    CONST robtarget T677:=[[56.500013,76.537078,6.249631],[1.000000,0.000000,0.000000,0.000000],[0,0,-1,0],[9E+09,9E+09,9E+09,9E+09,9E+09,9E+09]];
    CONST robtarget T678:=[[58.000019,76.384788,6.249631],[1.000000,0.000000,0.000000,0.000000],[0,0,-1,0],[9E+09,9E+09,9E+09,9E+09,9E+09,9E+09]];
    CONST robtarget T679:=[[58.000019,35.406248,6.249631],[1.000000,0.000000,0.000000,0.000000],[0,0,-1,0],[9E+09,9E+09,9E+09,9E+09,9E+09,9E+09]];
    CONST robtarget T680:=[[59.500025,35.473840,6.249631],[1.000000,0.000000,0.000000,0.000000],[0,0,-1,0],[9E+09,9E+09,9E+09,9E+09,9E+09,9E+09]];
    CONST robtarget T681:=[[59.500025,76.264330,6.249631],[1.000000,0.000000,0.000000,0.000000],[0,0,-1,0],[9E+09,9E+09,9E+09,9E+09,9E+09,9E+09]];
    CONST robtarget T682:=[[61.000031,76.089981,6.249631],[1.000000,0.000000,0.000000,0.000000],[0,0,-1,0],[9E+09,9E+09,9E+09,9E+09,9E+09,9E+09]];
    CONST robtarget T683:=[[61.000031,35.612525,6.249631],[1.000000,0.000000,0.000000,0.000000],[0,0,-1,0],[9E+09,9E+09,9E+09,9E+09,9E+09,9E+09]];
    CONST robtarget T684:=[[62.500037,35.829098,6.249631],[1.000000,0.000000,0.000000,0.000000],[0,0,-1,0],[9E+09,9E+09,9E+09,9E+09,9E+09,9E+09]];
    CONST robtarget T685:=[[62.500037,75.849994,6.249631],[1.000000,0.000000,0.000000,0.000000],[0,0,-1,0],[9E+09,9E+09,9E+09,9E+09,9E+09,9E+09]];
    CONST robtarget T686:=[[64.000043,75.305600,6.249631],[1.000000,0.000000,0.000000,0.000000],[0,0,-1,0],[9E+09,9E+09,9E+09,9E+09,9E+09,9E+09]];
    CONST robtarget T687:=[[64.000043,36.214677,6.249631],[1.000000,0.000000,0.000000,0.000000],[0,0,-1,0],[9E+09,9E+09,9E+09,9E+09,9E+09,9E+09]];
    CONST robtarget T688:=[[65.500049,36.567546,6.249631],[1.000000,0.000000,0.000000,0.000000],[0,0,-1,0],[9E+09,9E+09,9E+09,9E+09,9E+09,9E+09]];
    CONST robtarget T689:=[[65.500049,74.486668,6.249631],[1.000000,0.000000,0.000000,0.000000],[0,0,-1,0],[9E+09,9E+09,9E+09,9E+09,9E+09,9E+09]];
    CONST robtarget T690:=[[67.000055,73.456702,6.249631],[1.000000,0.000000,0.000000,0.000000],[0,0,-1,0],[9E+09,9E+09,9E+09,9E+09,9E+09,9E+09]];
    CONST robtarget T691:=[[67.000055,37.225942,6.249631],[1.000000,0.000000,0.000000,0.000000],[0,0,-1,0],[9E+09,9E+09,9E+09,9E+09,9E+09,9E+09]];
    CONST robtarget T692:=[[68.500061,37.908304,6.249631],[1.000000,0.000000,0.000000,0.000000],[0,0,-1,0],[9E+09,9E+09,9E+09,9E+09,9E+09,9E+09]];
    CONST robtarget T693:=[[68.500061,72.303444,6.249631],[1.000000,0.000000,0.000000,0.000000],[0,0,-1,0],[9E+09,9E+09,9E+09,9E+09,9E+09,9E+09]];
    CONST robtarget T694:=[[70.000067,70.867702,6.249631],[1.000000,0.000000,0.000000,0.000000],[0,0,-1,0],[9E+09,9E+09,9E+09,9E+09,9E+09,9E+09]];
    CONST robtarget T695:=[[70.000067,38.836205,6.249631],[1.000000,0.000000,0.000000,0.000000],[0,0,-1,0],[9E+09,9E+09,9E+09,9E+09,9E+09,9E+09]];
    CONST robtarget T696:=[[71.500073,39.891103,6.249631],[1.000000,0.000000,0.000000,0.000000],[0,0,-1,0],[9E+09,9E+09,9E+09,9E+09,9E+09,9E+09]];
    CONST robtarget T697:=[[71.500073,69.078100,6.249631],[1.000000,0.000000,0.000000,0.000000],[0,0,-1,0],[9E+09,9E+09,9E+09,9E+09,9E+09,9E+09]];
    CONST robtarget T698:=[[73.000079,66.945059,6.249631],[1.000000,0.000000,0.000000,0.000000],[0,0,-1,0],[9E+09,9E+09,9E+09,9E+09,9E+09,9E+09]];
    CONST robtarget T699:=[[73.000079,41.103881,6.249631],[1.000000,0.000000,0.000000,0.000000],[0,0,-1,0],[9E+09,9E+09,9E+09,9E+09,9E+09,9E+09]];
    CONST robtarget T700:=[[74.500085,42.494022,6.249631],[1.000000,0.000000,0.000000,0.000000],[0,0,-1,0],[9E+09,9E+09,9E+09,9E+09,9E+09,9E+09]];
    CONST robtarget T701:=[[74.500085,64.388687,6.249631],[1.000000,0.000000,0.000000,0.000000],[0,0,-1,0],[9E+09,9E+09,9E+09,9E+09,9E+09,9E+09]];
    CONST robtarget T702:=[[76.000091,60.363543,6.249631],[1.000000,0.000000,0.000000,0.000000],[0,0,-1,0],[9E+09,9E+09,9E+09,9E+09,9E+09,9E+09]];
    CONST robtarget T703:=[[76.000091,44.225148,6.249631],[1.000000,0.000000,0.000000,0.000000],[0,0,-1,0],[9E+09,9E+09,9E+09,9E+09,9E+09,9E+09]];
    CONST robtarget T704:=[[77.500097,47.712288,6.249631],[1.000000,0.000000,0.000000,0.000000],[0,0,-1,0],[9E+09,9E+09,9E+09,9E+09,9E+09,9E+09]];
    CONST robtarget T705:=[[77.500097,54.837844,6.249631],[1.000000,0.000000,0.000000,0.000000],[0,0,-1,0],[9E+09,9E+09,9E+09,9E+09,9E+09,9E+09]];
    CONST robtarget T706:=[[77.500097,46.672683,6.749641],[1.000000,0.000000,0.000000,0.000000],[0,0,-1,0],[9E+09,9E+09,9E+09,9E+09,9E+09,9E+09]];
    CONST robtarget T707:=[[77.500097,56.264594,6.749641],[1.000000,0.000000,0.000000,0.000000],[0,0,-1,0],[9E+09,9E+09,9E+09,9E+09,9E+09,9E+09]];
    CONST robtarget T708:=[[77.500097,46.672683,6.749641],[1.000000,0.000000,0.000000,0.000000],[0,0,-1,0],[9E+09,9E+09,9E+09,9E+09,9E+09,9E+09]];
    CONST robtarget T709:=[[77.500097,56.264594,6.749641],[1.000000,0.000000,0.000000,0.000000],[0,0,-1,0],[9E+09,9E+09,9E+09,9E+09,9E+09,9E+09]];
    CONST robtarget T710:=[[76.000091,60.945739,6.749641],[1.000000,0.000000,0.000000,0.000000],[0,0,-1,0],[9E+09,9E+09,9E+09,9E+09,9E+09,9E+09]];
    CONST robtarget T711:=[[76.000091,43.718418,6.749641],[1.000000,0.000000,0.000000,0.000000],[0,0,-1,0],[9E+09,9E+09,9E+09,9E+09,9E+09,9E+09]];
    CONST robtarget T712:=[[74.500085,42.018319,6.749641],[1.000000,0.000000,0.000000,0.000000],[0,0,-1,0],[9E+09,9E+09,9E+09,9E+09,9E+09,9E+09]];
    CONST robtarget T713:=[[74.500085,64.686211,6.749641],[1.000000,0.000000,0.000000,0.000000],[0,0,-1,0],[9E+09,9E+09,9E+09,9E+09,9E+09,9E+09]];
    CONST robtarget T714:=[[73.000079,67.110705,6.749641],[1.000000,0.000000,0.000000,0.000000],[0,0,-1,0],[9E+09,9E+09,9E+09,9E+09,9E+09,9E+09]];
    CONST robtarget T715:=[[73.000079,40.678790,6.749641],[1.000000,0.000000,0.000000,0.000000],[0,0,-1,0],[9E+09,9E+09,9E+09,9E+09,9E+09,9E+09]];
    CONST robtarget T716:=[[71.500073,39.412409,6.749641],[1.000000,0.000000,0.000000,0.000000],[0,0,-1,0],[9E+09,9E+09,9E+09,9E+09,9E+09,9E+09]];
    CONST robtarget T717:=[[71.500073,69.236494,6.749641],[1.000000,0.000000,0.000000,0.000000],[0,0,-1,0],[9E+09,9E+09,9E+09,9E+09,9E+09,9E+09]];
    CONST robtarget T718:=[[70.000067,71.090670,6.749641],[1.000000,0.000000,0.000000,0.000000],[0,0,-1,0],[9E+09,9E+09,9E+09,9E+09,9E+09,9E+09]];
    CONST robtarget T719:=[[70.000067,38.385338,6.749641],[1.000000,0.000000,0.000000,0.000000],[0,0,-1,0],[9E+09,9E+09,9E+09,9E+09,9E+09,9E+09]];
    CONST robtarget T720:=[[68.500061,37.449765,6.749641],[1.000000,0.000000,0.000000,0.000000],[0,0,-1,0],[9E+09,9E+09,9E+09,9E+09,9E+09,9E+09]];
    CONST robtarget T721:=[[68.500061,72.617147,6.749641],[1.000000,0.000000,0.000000,0.000000],[0,0,-1,0],[9E+09,9E+09,9E+09,9E+09,9E+09,9E+09]];
    CONST robtarget T722:=[[67.000055,73.796696,6.749641],[1.000000,0.000000,0.000000,0.000000],[0,0,-1,0],[9E+09,9E+09,9E+09,9E+09,9E+09,9E+09]];
    CONST robtarget T723:=[[67.000055,36.779468,6.749641],[1.000000,0.000000,0.000000,0.000000],[0,0,-1,0],[9E+09,9E+09,9E+09,9E+09,9E+09,9E+09]];
    CONST robtarget T724:=[[65.500049,36.130056,6.749641],[1.000000,0.000000,0.000000,0.000000],[0,0,-1,0],[9E+09,9E+09,9E+09,9E+09,9E+09,9E+09]];
    CONST robtarget T725:=[[65.500049,74.800360,6.749641],[1.000000,0.000000,0.000000,0.000000],[0,0,-1,0],[9E+09,9E+09,9E+09,9E+09,9E+09,9E+09]];
    CONST robtarget T726:=[[64.000043,75.578750,6.749641],[1.000000,0.000000,0.000000,0.000000],[0,0,-1,0],[9E+09,9E+09,9E+09,9E+09,9E+09,9E+09]];
    CONST robtarget T727:=[[64.000043,35.777188,6.749641],[1.000000,0.000000,0.000000,0.000000],[0,0,-1,0],[9E+09,9E+09,9E+09,9E+09,9E+09,9E+09]];
    CONST robtarget T728:=[[62.500037,35.412563,6.749641],[1.000000,0.000000,0.000000,0.000000],[0,0,-1,0],[9E+09,9E+09,9E+09,9E+09,9E+09,9E+09]];
    CONST robtarget T729:=[[62.500037,76.134604,6.749641],[1.000000,0.000000,0.000000,0.000000],[0,0,-1,0],[9E+09,9E+09,9E+09,9E+09,9E+09,9E+09]];
    CONST robtarget T730:=[[61.000031,76.390171,6.749641],[1.000000,0.000000,0.000000,0.000000],[0,0,-1,0],[9E+09,9E+09,9E+09,9E+09,9E+09,9E+09]];
    CONST robtarget T731:=[[61.000031,35.224978,6.749641],[1.000000,0.000000,0.000000,0.000000],[0,0,-1,0],[9E+09,9E+09,9E+09,9E+09,9E+09,9E+09]];
    CONST robtarget T732:=[[59.500025,35.088916,6.749641],[1.000000,0.000000,0.000000,0.000000],[0,0,-1,0],[9E+09,9E+09,9E+09,9E+09,9E+09,9E+09]];
    CONST robtarget T733:=[[59.500025,76.568137,6.749641],[1.000000,0.000000,0.000000,0.000000],[0,0,-1,0],[9E+09,9E+09,9E+09,9E+09,9E+09,9E+09]];
    CONST robtarget T734:=[[58.000019,76.697078,6.749641],[1.000000,0.000000,0.000000,0.000000],[0,0,-1,0],[9E+09,9E+09,9E+09,9E+09,9E+09,9E+09]];
    CONST robtarget T735:=[[58.000019,35.030106,6.749641],[1.000000,0.000000,0.000000,0.000000],[0,0,-1,0],[9E+09,9E+09,9E+09,9E+09,9E+09,9E+09]];
    CONST robtarget T736:=[[56.500013,34.993140,6.749641],[1.000000,0.000000,0.000000,0.000000],[0,0,-1,0],[9E+09,9E+09,9E+09,9E+09,9E+09,9E+09]];
    CONST robtarget T737:=[[56.500013,76.858293,6.749641],[1.000000,0.000000,0.000000,0.000000],[0,0,-1,0],[9E+09,9E+09,9E+09,9E+09,9E+09,9E+09]];
    CONST robtarget T738:=[[55.000007,76.963959,6.749641],[1.000000,0.000000,0.000000,0.000000],[0,0,-1,0],[9E+09,9E+09,9E+09,9E+09,9E+09,9E+09]];
    CONST robtarget T739:=[[55.000007,34.997342,6.749641],[1.000000,0.000000,0.000000,0.000000],[0,0,-1,0],[9E+09,9E+09,9E+09,9E+09,9E+09,9E+09]];
    CONST robtarget T740:=[[53.500001,34.993140,6.749641],[1.000000,0.000000,0.000000,0.000000],[0,0,-1,0],[9E+09,9E+09,9E+09,9E+09,9E+09,9E+09]];
    CONST robtarget T741:=[[53.500001,76.858293,6.749641],[1.000000,0.000000,0.000000,0.000000],[0,0,-1,0],[9E+09,9E+09,9E+09,9E+09,9E+09,9E+09]];
    CONST robtarget T742:=[[51.999995,76.697078,6.749641],[1.000000,0.000000,0.000000,0.000000],[0,0,-1,0],[9E+09,9E+09,9E+09,9E+09,9E+09,9E+09]];
    CONST robtarget T743:=[[51.999995,35.030107,6.749641],[1.000000,0.000000,0.000000,0.000000],[0,0,-1,0],[9E+09,9E+09,9E+09,9E+09,9E+09,9E+09]];
    CONST robtarget T744:=[[50.499989,35.088916,6.749641],[1.000000,0.000000,0.000000,0.000000],[0,0,-1,0],[9E+09,9E+09,9E+09,9E+09,9E+09,9E+09]];
    CONST robtarget T745:=[[50.499989,76.568136,6.749641],[1.000000,0.000000,0.000000,0.000000],[0,0,-1,0],[9E+09,9E+09,9E+09,9E+09,9E+09,9E+09]];
    CONST robtarget T746:=[[48.999983,76.390167,6.749641],[1.000000,0.000000,0.000000,0.000000],[0,0,-1,0],[9E+09,9E+09,9E+09,9E+09,9E+09,9E+09]];
    CONST robtarget T747:=[[48.999983,35.224979,6.749641],[1.000000,0.000000,0.000000,0.000000],[0,0,-1,0],[9E+09,9E+09,9E+09,9E+09,9E+09,9E+09]];
    CONST robtarget T748:=[[47.499977,35.412564,6.749641],[1.000000,0.000000,0.000000,0.000000],[0,0,-1,0],[9E+09,9E+09,9E+09,9E+09,9E+09,9E+09]];
    CONST robtarget T749:=[[47.499977,76.134597,6.749641],[1.000000,0.000000,0.000000,0.000000],[0,0,-1,0],[9E+09,9E+09,9E+09,9E+09,9E+09,9E+09]];
    CONST robtarget T750:=[[45.999971,75.578745,6.749641],[1.000000,0.000000,0.000000,0.000000],[0,0,-1,0],[9E+09,9E+09,9E+09,9E+09,9E+09,9E+09]];
    CONST robtarget T751:=[[45.999971,35.777189,6.749641],[1.000000,0.000000,0.000000,0.000000],[0,0,-1,0],[9E+09,9E+09,9E+09,9E+09,9E+09,9E+09]];
    CONST robtarget T752:=[[44.499965,36.130058,6.749641],[1.000000,0.000000,0.000000,0.000000],[0,0,-1,0],[9E+09,9E+09,9E+09,9E+09,9E+09,9E+09]];
    CONST robtarget T753:=[[44.499965,74.800359,6.749641],[1.000000,0.000000,0.000000,0.000000],[0,0,-1,0],[9E+09,9E+09,9E+09,9E+09,9E+09,9E+09]];
    CONST robtarget T754:=[[42.999959,73.796696,6.749641],[1.000000,0.000000,0.000000,0.000000],[0,0,-1,0],[9E+09,9E+09,9E+09,9E+09,9E+09,9E+09]];
    CONST robtarget T755:=[[42.999959,36.779470,6.749641],[1.000000,0.000000,0.000000,0.000000],[0,0,-1,0],[9E+09,9E+09,9E+09,9E+09,9E+09,9E+09]];
    CONST robtarget T756:=[[41.499953,37.449766,6.749641],[1.000000,0.000000,0.000000,0.000000],[0,0,-1,0],[9E+09,9E+09,9E+09,9E+09,9E+09,9E+09]];
    CONST robtarget T757:=[[41.499953,72.617146,6.749641],[1.000000,0.000000,0.000000,0.000000],[0,0,-1,0],[9E+09,9E+09,9E+09,9E+09,9E+09,9E+09]];
    CONST robtarget T758:=[[39.999947,71.090670,6.749641],[1.000000,0.000000,0.000000,0.000000],[0,0,-1,0],[9E+09,9E+09,9E+09,9E+09,9E+09,9E+09]];
    CONST robtarget T759:=[[39.999947,38.385339,6.749641],[1.000000,0.000000,0.000000,0.000000],[0,0,-1,0],[9E+09,9E+09,9E+09,9E+09,9E+09,9E+09]];
    CONST robtarget T760:=[[38.499941,39.412415,6.749641],[1.000000,0.000000,0.000000,0.000000],[0,0,-1,0],[9E+09,9E+09,9E+09,9E+09,9E+09,9E+09]];
    CONST robtarget T761:=[[38.499941,69.236494,6.749641],[1.000000,0.000000,0.000000,0.000000],[0,0,-1,0],[9E+09,9E+09,9E+09,9E+09,9E+09,9E+09]];
    CONST robtarget T762:=[[36.999935,67.112770,6.749641],[1.000000,0.000000,0.000000,0.000000],[0,0,-1,0],[9E+09,9E+09,9E+09,9E+09,9E+09,9E+09]];
    CONST robtarget T763:=[[36.999935,40.678790,6.749641],[1.000000,0.000000,0.000000,0.000000],[0,0,-1,0],[9E+09,9E+09,9E+09,9E+09,9E+09,9E+09]];
    CONST robtarget T764:=[[35.499929,42.018319,6.749641],[1.000000,0.000000,0.000000,0.000000],[0,0,-1,0],[9E+09,9E+09,9E+09,9E+09,9E+09,9E+09]];
    CONST robtarget T765:=[[35.499929,64.692749,6.749641],[1.000000,0.000000,0.000000,0.000000],[0,0,-1,0],[9E+09,9E+09,9E+09,9E+09,9E+09,9E+09]];
    CONST robtarget T766:=[[33.999923,60.962386,6.749641],[1.000000,0.000000,0.000000,0.000000],[0,0,-1,0],[9E+09,9E+09,9E+09,9E+09,9E+09,9E+09]];
    CONST robtarget T767:=[[33.999923,43.718418,6.749641],[1.000000,0.000000,0.000000,0.000000],[0,0,-1,0],[9E+09,9E+09,9E+09,9E+09,9E+09,9E+09]];
    CONST robtarget T768:=[[32.499917,46.672683,6.749641],[1.000000,0.000000,0.000000,0.000000],[0,0,-1,0],[9E+09,9E+09,9E+09,9E+09,9E+09,9E+09]];
    CONST robtarget T769:=[[32.499917,56.267195,6.749641],[1.000000,0.000000,0.000000,0.000000],[0,0,-1,0],[9E+09,9E+09,9E+09,9E+09,9E+09,9E+09]];
    CONST robtarget T770:=[[31.749914,48.149744,7.249651],[1.000000,0.000000,0.000000,0.000000],[0,0,-1,0],[9E+09,9E+09,9E+09,9E+09,9E+09,9E+09]];
    CONST robtarget T771:=[[31.749914,55.186707,7.249651],[1.000000,0.000000,0.000000,0.000000],[0,0,-1,0],[9E+09,9E+09,9E+09,9E+09,9E+09,9E+09]];
    CONST robtarget T772:=[[31.749914,48.149744,7.249651],[1.000000,0.000000,0.000000,0.000000],[0,0,-1,0],[9E+09,9E+09,9E+09,9E+09,9E+09,9E+09]];
    CONST robtarget T773:=[[31.749914,55.186707,7.249651],[1.000000,0.000000,0.000000,0.000000],[0,0,-1,0],[9E+09,9E+09,9E+09,9E+09,9E+09,9E+09]];
    CONST robtarget T774:=[[33.249920,59.803507,7.249651],[1.000000,0.000000,0.000000,0.000000],[0,0,-1,0],[9E+09,9E+09,9E+09,9E+09,9E+09,9E+09]];
    CONST robtarget T775:=[[33.249920,44.412102,7.249651],[1.000000,0.000000,0.000000,0.000000],[0,0,-1,0],[9E+09,9E+09,9E+09,9E+09,9E+09,9E+09]];
    CONST robtarget T776:=[[34.749926,42.393779,7.249651],[1.000000,0.000000,0.000000,0.000000],[0,0,-1,0],[9E+09,9E+09,9E+09,9E+09,9E+09,9E+09]];
    CONST robtarget T777:=[[34.749926,63.502702,7.249651],[1.000000,0.000000,0.000000,0.000000],[0,0,-1,0],[9E+09,9E+09,9E+09,9E+09,9E+09,9E+09]];
    CONST robtarget T778:=[[36.249932,66.269036,7.249651],[1.000000,0.000000,0.000000,0.000000],[0,0,-1,0],[9E+09,9E+09,9E+09,9E+09,9E+09,9E+09]];
    CONST robtarget T779:=[[36.249932,40.845337,7.249651],[1.000000,0.000000,0.000000,0.000000],[0,0,-1,0],[9E+09,9E+09,9E+09,9E+09,9E+09,9E+09]];
    CONST robtarget T780:=[[37.749938,39.581246,7.249651],[1.000000,0.000000,0.000000,0.000000],[0,0,-1,0],[9E+09,9E+09,9E+09,9E+09,9E+09,9E+09]];
    CONST robtarget T781:=[[37.749938,68.403249,7.249651],[1.000000,0.000000,0.000000,0.000000],[0,0,-1,0],[9E+09,9E+09,9E+09,9E+09,9E+09,9E+09]];
    CONST robtarget T782:=[[39.249944,70.294316,7.249651],[1.000000,0.000000,0.000000,0.000000],[0,0,-1,0],[9E+09,9E+09,9E+09,9E+09,9E+09,9E+09]];
    CONST robtarget T783:=[[39.249944,38.419874,7.249651],[1.000000,0.000000,0.000000,0.000000],[0,0,-1,0],[9E+09,9E+09,9E+09,9E+09,9E+09,9E+09]];
    CONST robtarget T784:=[[40.749950,37.456690,7.249651],[1.000000,0.000000,0.000000,0.000000],[0,0,-1,0],[9E+09,9E+09,9E+09,9E+09,9E+09,9E+09]];
    CONST robtarget T785:=[[40.749950,72.153255,7.249651],[1.000000,0.000000,0.000000,0.000000],[0,0,-1,0],[9E+09,9E+09,9E+09,9E+09,9E+09,9E+09]];
    CONST robtarget T786:=[[42.249956,73.487604,7.249651],[1.000000,0.000000,0.000000,0.000000],[0,0,-1,0],[9E+09,9E+09,9E+09,9E+09,9E+09,9E+09]];
    CONST robtarget T787:=[[42.249956,36.665124,7.249651],[1.000000,0.000000,0.000000,0.000000],[0,0,-1,0],[9E+09,9E+09,9E+09,9E+09,9E+09,9E+09]];
    CONST robtarget T788:=[[43.749962,35.996740,7.249651],[1.000000,0.000000,0.000000,0.000000],[0,0,-1,0],[9E+09,9E+09,9E+09,9E+09,9E+09,9E+09]];
    CONST robtarget T789:=[[43.749962,74.595147,7.249651],[1.000000,0.000000,0.000000,0.000000],[0,0,-1,0],[9E+09,9E+09,9E+09,9E+09,9E+09,9E+09]];
    CONST robtarget T790:=[[45.249968,75.543611,7.249651],[1.000000,0.000000,0.000000,0.000000],[0,0,-1,0],[9E+09,9E+09,9E+09,9E+09,9E+09,9E+09]];
    CONST robtarget T791:=[[45.249968,35.516134,7.249651],[1.000000,0.000000,0.000000,0.000000],[0,0,-1,0],[9E+09,9E+09,9E+09,9E+09,9E+09,9E+09]];
    CONST robtarget T792:=[[46.749974,35.163265,7.249651],[1.000000,0.000000,0.000000,0.000000],[0,0,-1,0],[9E+09,9E+09,9E+09,9E+09,9E+09,9E+09]];
    CONST robtarget T793:=[[46.749974,76.146737,7.249651],[1.000000,0.000000,0.000000,0.000000],[0,0,-1,0],[9E+09,9E+09,9E+09,9E+09,9E+09,9E+09]];
    CONST robtarget T794:=[[48.249980,76.554434,7.249651],[1.000000,0.000000,0.000000,0.000000],[0,0,-1,0],[9E+09,9E+09,9E+09,9E+09,9E+09,9E+09]];
    CONST robtarget T795:=[[48.249980,34.917920,7.249651],[1.000000,0.000000,0.000000,0.000000],[0,0,-1,0],[9E+09,9E+09,9E+09,9E+09,9E+09,9E+09]];
    CONST robtarget T796:=[[49.749986,34.756945,7.249651],[1.000000,0.000000,0.000000,0.000000],[0,0,-1,0],[9E+09,9E+09,9E+09,9E+09,9E+09,9E+09]];
    CONST robtarget T797:=[[49.749986,76.806238,7.249651],[1.000000,0.000000,0.000000,0.000000],[0,0,-1,0],[9E+09,9E+09,9E+09,9E+09,9E+09,9E+09]];
    CONST robtarget T798:=[[51.249992,76.939585,7.249651],[1.000000,0.000000,0.000000,0.000000],[0,0,-1,0],[9E+09,9E+09,9E+09,9E+09,9E+09,9E+09]];
    CONST robtarget T799:=[[51.249992,34.674587,7.249651],[1.000000,0.000000,0.000000,0.000000],[0,0,-1,0],[9E+09,9E+09,9E+09,9E+09,9E+09,9E+09]];
    CONST robtarget T800:=[[52.749998,34.617779,7.249651],[1.000000,0.000000,0.000000,0.000000],[0,0,-1,0],[9E+09,9E+09,9E+09,9E+09,9E+09,9E+09]];
    CONST robtarget T801:=[[52.749998,77.095672,7.249651],[1.000000,0.000000,0.000000,0.000000],[0,0,-1,0],[9E+09,9E+09,9E+09,9E+09,9E+09,9E+09]];
    CONST robtarget T802:=[[54.250004,77.233300,7.249651],[1.000000,0.000000,0.000000,0.000000],[0,0,-1,0],[9E+09,9E+09,9E+09,9E+09,9E+09,9E+09]];
    CONST robtarget T803:=[[54.250004,34.621983,7.249651],[1.000000,0.000000,0.000000,0.000000],[0,0,-1,0],[9E+09,9E+09,9E+09,9E+09,9E+09,9E+09]];
    CONST robtarget T804:=[[55.750010,34.621983,7.249651],[1.000000,0.000000,0.000000,0.000000],[0,0,-1,0],[9E+09,9E+09,9E+09,9E+09,9E+09,9E+09]];
    CONST robtarget T805:=[[55.750010,77.233300,7.249651],[1.000000,0.000000,0.000000,0.000000],[0,0,-1,0],[9E+09,9E+09,9E+09,9E+09,9E+09,9E+09]];
    CONST robtarget T806:=[[57.250016,77.095672,7.249651],[1.000000,0.000000,0.000000,0.000000],[0,0,-1,0],[9E+09,9E+09,9E+09,9E+09,9E+09,9E+09]];
    CONST robtarget T807:=[[57.250016,34.617779,7.249651],[1.000000,0.000000,0.000000,0.000000],[0,0,-1,0],[9E+09,9E+09,9E+09,9E+09,9E+09,9E+09]];
    CONST robtarget T808:=[[58.750022,34.674587,7.249651],[1.000000,0.000000,0.000000,0.000000],[0,0,-1,0],[9E+09,9E+09,9E+09,9E+09,9E+09,9E+09]];
    CONST robtarget T809:=[[58.750022,76.939585,7.249651],[1.000000,0.000000,0.000000,0.000000],[0,0,-1,0],[9E+09,9E+09,9E+09,9E+09,9E+09,9E+09]];
    CONST robtarget T810:=[[60.250028,76.806238,7.249651],[1.000000,0.000000,0.000000,0.000000],[0,0,-1,0],[9E+09,9E+09,9E+09,9E+09,9E+09,9E+09]];
    CONST robtarget T811:=[[60.250028,34.756945,7.249651],[1.000000,0.000000,0.000000,0.000000],[0,0,-1,0],[9E+09,9E+09,9E+09,9E+09,9E+09,9E+09]];
    CONST robtarget T812:=[[61.750034,34.917920,7.249651],[1.000000,0.000000,0.000000,0.000000],[0,0,-1,0],[9E+09,9E+09,9E+09,9E+09,9E+09,9E+09]];
    CONST robtarget T813:=[[61.750034,76.554438,7.249651],[1.000000,0.000000,0.000000,0.000000],[0,0,-1,0],[9E+09,9E+09,9E+09,9E+09,9E+09,9E+09]];
    CONST robtarget T814:=[[63.250040,76.146743,7.249651],[1.000000,0.000000,0.000000,0.000000],[0,0,-1,0],[9E+09,9E+09,9E+09,9E+09,9E+09,9E+09]];
    CONST robtarget T815:=[[63.250040,35.163264,7.249651],[1.000000,0.000000,0.000000,0.000000],[0,0,-1,0],[9E+09,9E+09,9E+09,9E+09,9E+09,9E+09]];
    CONST robtarget T816:=[[64.750046,35.516132,7.249651],[1.000000,0.000000,0.000000,0.000000],[0,0,-1,0],[9E+09,9E+09,9E+09,9E+09,9E+09,9E+09]];
    CONST robtarget T817:=[[64.750046,75.543611,7.249651],[1.000000,0.000000,0.000000,0.000000],[0,0,-1,0],[9E+09,9E+09,9E+09,9E+09,9E+09,9E+09]];
    CONST robtarget T818:=[[66.250052,74.595146,7.249651],[1.000000,0.000000,0.000000,0.000000],[0,0,-1,0],[9E+09,9E+09,9E+09,9E+09,9E+09,9E+09]];
    CONST robtarget T819:=[[66.250052,35.996736,7.249651],[1.000000,0.000000,0.000000,0.000000],[0,0,-1,0],[9E+09,9E+09,9E+09,9E+09,9E+09,9E+09]];
    CONST robtarget T820:=[[67.750058,36.665123,7.249651],[1.000000,0.000000,0.000000,0.000000],[0,0,-1,0],[9E+09,9E+09,9E+09,9E+09,9E+09,9E+09]];
    CONST robtarget T821:=[[67.750058,73.487604,7.249651],[1.000000,0.000000,0.000000,0.000000],[0,0,-1,0],[9E+09,9E+09,9E+09,9E+09,9E+09,9E+09]];
    CONST robtarget T822:=[[69.250064,72.153254,7.249651],[1.000000,0.000000,0.000000,0.000000],[0,0,-1,0],[9E+09,9E+09,9E+09,9E+09,9E+09,9E+09]];
    CONST robtarget T823:=[[69.250064,37.456690,7.249651],[1.000000,0.000000,0.000000,0.000000],[0,0,-1,0],[9E+09,9E+09,9E+09,9E+09,9E+09,9E+09]];
    CONST robtarget T824:=[[70.750070,38.419869,7.249651],[1.000000,0.000000,0.000000,0.000000],[0,0,-1,0],[9E+09,9E+09,9E+09,9E+09,9E+09,9E+09]];
    CONST robtarget T825:=[[70.750070,70.294314,7.249651],[1.000000,0.000000,0.000000,0.000000],[0,0,-1,0],[9E+09,9E+09,9E+09,9E+09,9E+09,9E+09]];
    CONST robtarget T826:=[[72.250076,68.402546,7.249651],[1.000000,0.000000,0.000000,0.000000],[0,0,-1,0],[9E+09,9E+09,9E+09,9E+09,9E+09,9E+09]];
    CONST robtarget T827:=[[72.250076,39.581241,7.249651],[1.000000,0.000000,0.000000,0.000000],[0,0,-1,0],[9E+09,9E+09,9E+09,9E+09,9E+09,9E+09]];
    CONST robtarget T828:=[[73.750082,40.845337,7.249651],[1.000000,0.000000,0.000000,0.000000],[0,0,-1,0],[9E+09,9E+09,9E+09,9E+09,9E+09,9E+09]];
    CONST robtarget T829:=[[73.750082,66.267104,7.249651],[1.000000,0.000000,0.000000,0.000000],[0,0,-1,0],[9E+09,9E+09,9E+09,9E+09,9E+09,9E+09]];
    CONST robtarget T830:=[[75.250088,63.493217,7.249651],[1.000000,0.000000,0.000000,0.000000],[0,0,-1,0],[9E+09,9E+09,9E+09,9E+09,9E+09,9E+09]];
    CONST robtarget T831:=[[75.250088,42.393780,7.249651],[1.000000,0.000000,0.000000,0.000000],[0,0,-1,0],[9E+09,9E+09,9E+09,9E+09,9E+09,9E+09]];
    CONST robtarget T832:=[[76.750094,44.412104,7.249651],[1.000000,0.000000,0.000000,0.000000],[0,0,-1,0],[9E+09,9E+09,9E+09,9E+09,9E+09,9E+09]];
    CONST robtarget T833:=[[76.750094,59.798561,7.249651],[1.000000,0.000000,0.000000,0.000000],[0,0,-1,0],[9E+09,9E+09,9E+09,9E+09,9E+09,9E+09]];
    CONST robtarget T834:=[[78.250100,55.186221,7.249651],[1.000000,0.000000,0.000000,0.000000],[0,0,-1,0],[9E+09,9E+09,9E+09,9E+09,9E+09,9E+09]];
    CONST robtarget T835:=[[78.250100,48.149743,7.249651],[1.000000,0.000000,0.000000,0.000000],[0,0,-1,0],[9E+09,9E+09,9E+09,9E+09,9E+09,9E+09]];
    CONST robtarget T836:=[[78.250100,47.245248,7.749661],[1.000000,0.000000,0.000000,0.000000],[0,0,-1,0],[9E+09,9E+09,9E+09,9E+09,9E+09,9E+09]];
    CONST robtarget T837:=[[78.250100,56.662837,7.749661],[1.000000,0.000000,0.000000,0.000000],[0,0,-1,0],[9E+09,9E+09,9E+09,9E+09,9E+09,9E+09]];
    CONST robtarget T838:=[[78.250100,47.245248,7.749661],[1.000000,0.000000,0.000000,0.000000],[0,0,-1,0],[9E+09,9E+09,9E+09,9E+09,9E+09,9E+09]];
    CONST robtarget T839:=[[78.250100,56.662837,7.749661],[1.000000,0.000000,0.000000,0.000000],[0,0,-1,0],[9E+09,9E+09,9E+09,9E+09,9E+09,9E+09]];
    CONST robtarget T840:=[[76.750094,60.836207,7.749661],[1.000000,0.000000,0.000000,0.000000],[0,0,-1,0],[9E+09,9E+09,9E+09,9E+09,9E+09,9E+09]];
    CONST robtarget T841:=[[76.750094,43.798340,7.749661],[1.000000,0.000000,0.000000,0.000000],[0,0,-1,0],[9E+09,9E+09,9E+09,9E+09,9E+09,9E+09]];
    CONST robtarget T842:=[[75.250088,41.935067,7.749661],[1.000000,0.000000,0.000000,0.000000],[0,0,-1,0],[9E+09,9E+09,9E+09,9E+09,9E+09,9E+09]];
    CONST robtarget T843:=[[75.250088,63.787391,7.749661],[1.000000,0.000000,0.000000,0.000000],[0,0,-1,0],[9E+09,9E+09,9E+09,9E+09,9E+09,9E+09]];
    CONST robtarget T844:=[[73.750082,66.460200,7.749661],[1.000000,0.000000,0.000000,0.000000],[0,0,-1,0],[9E+09,9E+09,9E+09,9E+09,9E+09,9E+09]];
    CONST robtarget T845:=[[73.750082,40.397598,7.749661],[1.000000,0.000000,0.000000,0.000000],[0,0,-1,0],[9E+09,9E+09,9E+09,9E+09,9E+09,9E+09]];
    CONST robtarget T846:=[[72.250076,39.102547,7.749661],[1.000000,0.000000,0.000000,0.000000],[0,0,-1,0],[9E+09,9E+09,9E+09,9E+09,9E+09,9E+09]];
    CONST robtarget T847:=[[72.250076,68.562468,7.749661],[1.000000,0.000000,0.000000,0.000000],[0,0,-1,0],[9E+09,9E+09,9E+09,9E+09,9E+09,9E+09]];
    CONST robtarget T848:=[[70.750070,70.517281,7.749661],[1.000000,0.000000,0.000000,0.000000],[0,0,-1,0],[9E+09,9E+09,9E+09,9E+09,9E+09,9E+09]];
    CONST robtarget T849:=[[70.750070,37.972811,7.749661],[1.000000,0.000000,0.000000,0.000000],[0,0,-1,0],[9E+09,9E+09,9E+09,9E+09,9E+09,9E+09]];
    CONST robtarget T850:=[[69.250064,37.009631,7.749661],[1.000000,0.000000,0.000000,0.000000],[0,0,-1,0],[9E+09,9E+09,9E+09,9E+09,9E+09,9E+09]];
    CONST robtarget T851:=[[69.250064,72.379154,7.749661],[1.000000,0.000000,0.000000,0.000000],[0,0,-1,0],[9E+09,9E+09,9E+09,9E+09,9E+09,9E+09]];
    CONST robtarget T852:=[[67.750058,73.752852,7.749661],[1.000000,0.000000,0.000000,0.000000],[0,0,-1,0],[9E+09,9E+09,9E+09,9E+09,9E+09,9E+09]];
    CONST robtarget T853:=[[67.750058,36.216809,7.749661],[1.000000,0.000000,0.000000,0.000000],[0,0,-1,0],[9E+09,9E+09,9E+09,9E+09,9E+09,9E+09]];
    CONST robtarget T854:=[[66.250052,35.600952,7.749661],[1.000000,0.000000,0.000000,0.000000],[0,0,-1,0],[9E+09,9E+09,9E+09,9E+09,9E+09,9E+09]];
    CONST robtarget T855:=[[66.250052,74.877969,7.749661],[1.000000,0.000000,0.000000,0.000000],[0,0,-1,0],[9E+09,9E+09,9E+09,9E+09,9E+09,9E+09]];
    CONST robtarget T856:=[[64.750046,75.808847,7.749661],[1.000000,0.000000,0.000000,0.000000],[0,0,-1,0],[9E+09,9E+09,9E+09,9E+09,9E+09,9E+09]];
    CONST robtarget T857:=[[64.750046,35.162829,7.749661],[1.000000,0.000000,0.000000,0.000000],[0,0,-1,0],[9E+09,9E+09,9E+09,9E+09,9E+09,9E+09]];
    CONST robtarget T858:=[[63.250040,34.832357,7.749661],[1.000000,0.000000,0.000000,0.000000],[0,0,-1,0],[9E+09,9E+09,9E+09,9E+09,9E+09,9E+09]];
    CONST robtarget T859:=[[63.250040,76.419230,7.749661],[1.000000,0.000000,0.000000,0.000000],[0,0,-1,0],[9E+09,9E+09,9E+09,9E+09,9E+09,9E+09]];
    CONST robtarget T860:=[[61.750034,76.839048,7.749661],[1.000000,0.000000,0.000000,0.000000],[0,0,-1,0],[9E+09,9E+09,9E+09,9E+09,9E+09,9E+09]];
    CONST robtarget T861:=[[61.750034,34.619021,7.749661],[1.000000,0.000000,0.000000,0.000000],[0,0,-1,0],[9E+09,9E+09,9E+09,9E+09,9E+09,9E+09]];
    CONST robtarget T862:=[[60.250028,34.461894,7.749661],[1.000000,0.000000,0.000000,0.000000],[0,0,-1,0],[9E+09,9E+09,9E+09,9E+09,9E+09,9E+09]];
    CONST robtarget T863:=[[60.250028,77.106429,7.749661],[1.000000,0.000000,0.000000,0.000000],[0,0,-1,0],[9E+09,9E+09,9E+09,9E+09,9E+09,9E+09]];
    CONST robtarget T864:=[[58.750022,77.251875,7.749661],[1.000000,0.000000,0.000000,0.000000],[0,0,-1,0],[9E+09,9E+09,9E+09,9E+09,9E+09,9E+09]];
    CONST robtarget T865:=[[58.750022,34.377538,7.749661],[1.000000,0.000000,0.000000,0.000000],[0,0,-1,0],[9E+09,9E+09,9E+09,9E+09,9E+09,9E+09]];
    CONST robtarget T866:=[[57.250016,34.317308,7.749661],[1.000000,0.000000,0.000000,0.000000],[0,0,-1,0],[9E+09,9E+09,9E+09,9E+09,9E+09,9E+09]];
    CONST robtarget T867:=[[57.250016,77.407458,7.749661],[1.000000,0.000000,0.000000,0.000000],[0,0,-1,0],[9E+09,9E+09,9E+09,9E+09,9E+09,9E+09]];
    CONST robtarget T868:=[[55.750010,77.559108,7.749661],[1.000000,0.000000,0.000000,0.000000],[0,0,-1,0],[9E+09,9E+09,9E+09,9E+09,9E+09,9E+09]];
    CONST robtarget T869:=[[55.750010,34.318112,7.749661],[1.000000,0.000000,0.000000,0.000000],[0,0,-1,0],[9E+09,9E+09,9E+09,9E+09,9E+09,9E+09]];
    CONST robtarget T870:=[[54.250004,34.318112,7.749661],[1.000000,0.000000,0.000000,0.000000],[0,0,-1,0],[9E+09,9E+09,9E+09,9E+09,9E+09,9E+09]];
    CONST robtarget T871:=[[54.250004,77.559108,7.749661],[1.000000,0.000000,0.000000,0.000000],[0,0,-1,0],[9E+09,9E+09,9E+09,9E+09,9E+09,9E+09]];
    CONST robtarget T872:=[[52.749998,77.407458,7.749661],[1.000000,0.000000,0.000000,0.000000],[0,0,-1,0],[9E+09,9E+09,9E+09,9E+09,9E+09,9E+09]];
    CONST robtarget T873:=[[52.749998,34.317308,7.749661],[1.000000,0.000000,0.000000,0.000000],[0,0,-1,0],[9E+09,9E+09,9E+09,9E+09,9E+09,9E+09]];
    CONST robtarget T874:=[[51.249992,34.377538,7.749661],[1.000000,0.000000,0.000000,0.000000],[0,0,-1,0],[9E+09,9E+09,9E+09,9E+09,9E+09,9E+09]];
    CONST robtarget T875:=[[51.249992,77.251875,7.749661],[1.000000,0.000000,0.000000,0.000000],[0,0,-1,0],[9E+09,9E+09,9E+09,9E+09,9E+09,9E+09]];
    CONST robtarget T876:=[[49.749986,77.106428,7.749661],[1.000000,0.000000,0.000000,0.000000],[0,0,-1,0],[9E+09,9E+09,9E+09,9E+09,9E+09,9E+09]];
    CONST robtarget T877:=[[49.749986,34.461894,7.749661],[1.000000,0.000000,0.000000,0.000000],[0,0,-1,0],[9E+09,9E+09,9E+09,9E+09,9E+09,9E+09]];
    CONST robtarget T878:=[[48.249980,34.619021,7.749661],[1.000000,0.000000,0.000000,0.000000],[0,0,-1,0],[9E+09,9E+09,9E+09,9E+09,9E+09,9E+09]];
    CONST robtarget T879:=[[48.249980,76.839046,7.749661],[1.000000,0.000000,0.000000,0.000000],[0,0,-1,0],[9E+09,9E+09,9E+09,9E+09,9E+09,9E+09]];
    CONST robtarget T880:=[[46.749974,76.419228,7.749661],[1.000000,0.000000,0.000000,0.000000],[0,0,-1,0],[9E+09,9E+09,9E+09,9E+09,9E+09,9E+09]];
    CONST robtarget T881:=[[46.749974,34.832358,7.749661],[1.000000,0.000000,0.000000,0.000000],[0,0,-1,0],[9E+09,9E+09,9E+09,9E+09,9E+09,9E+09]];
    CONST robtarget T882:=[[45.249968,35.162831,7.749661],[1.000000,0.000000,0.000000,0.000000],[0,0,-1,0],[9E+09,9E+09,9E+09,9E+09,9E+09,9E+09]];
    CONST robtarget T883:=[[45.249968,75.808848,7.749661],[1.000000,0.000000,0.000000,0.000000],[0,0,-1,0],[9E+09,9E+09,9E+09,9E+09,9E+09,9E+09]];
    CONST robtarget T884:=[[43.749962,74.877970,7.749661],[1.000000,0.000000,0.000000,0.000000],[0,0,-1,0],[9E+09,9E+09,9E+09,9E+09,9E+09,9E+09]];
    CONST robtarget T885:=[[43.749962,35.600956,7.749661],[1.000000,0.000000,0.000000,0.000000],[0,0,-1,0],[9E+09,9E+09,9E+09,9E+09,9E+09,9E+09]];
    CONST robtarget T886:=[[42.249956,36.216811,7.749661],[1.000000,0.000000,0.000000,0.000000],[0,0,-1,0],[9E+09,9E+09,9E+09,9E+09,9E+09,9E+09]];
    CONST robtarget T887:=[[42.249956,73.752852,7.749661],[1.000000,0.000000,0.000000,0.000000],[0,0,-1,0],[9E+09,9E+09,9E+09,9E+09,9E+09,9E+09]];
    CONST robtarget T888:=[[40.749950,72.379155,7.749661],[1.000000,0.000000,0.000000,0.000000],[0,0,-1,0],[9E+09,9E+09,9E+09,9E+09,9E+09,9E+09]];
    CONST robtarget T889:=[[40.749950,37.009633,7.749661],[1.000000,0.000000,0.000000,0.000000],[0,0,-1,0],[9E+09,9E+09,9E+09,9E+09,9E+09,9E+09]];
    CONST robtarget T890:=[[39.249944,37.972818,7.749661],[1.000000,0.000000,0.000000,0.000000],[0,0,-1,0],[9E+09,9E+09,9E+09,9E+09,9E+09,9E+09]];
    CONST robtarget T891:=[[39.249944,70.517283,7.749661],[1.000000,0.000000,0.000000,0.000000],[0,0,-1,0],[9E+09,9E+09,9E+09,9E+09,9E+09,9E+09]];
    CONST robtarget T892:=[[37.749938,68.563162,7.749661],[1.000000,0.000000,0.000000,0.000000],[0,0,-1,0],[9E+09,9E+09,9E+09,9E+09,9E+09,9E+09]];
    CONST robtarget T893:=[[37.749938,39.102555,7.749661],[1.000000,0.000000,0.000000,0.000000],[0,0,-1,0],[9E+09,9E+09,9E+09,9E+09,9E+09,9E+09]];
    CONST robtarget T894:=[[36.249932,40.397599,7.749661],[1.000000,0.000000,0.000000,0.000000],[0,0,-1,0],[9E+09,9E+09,9E+09,9E+09,9E+09,9E+09]];
    CONST robtarget T895:=[[36.249932,66.461721,7.749661],[1.000000,0.000000,0.000000,0.000000],[0,0,-1,0],[9E+09,9E+09,9E+09,9E+09,9E+09,9E+09]];
    CONST robtarget T896:=[[34.749926,63.785052,7.749661],[1.000000,0.000000,0.000000,0.000000],[0,0,-1,0],[9E+09,9E+09,9E+09,9E+09,9E+09,9E+09]];
    CONST robtarget T897:=[[34.749926,41.935066,7.749661],[1.000000,0.000000,0.000000,0.000000],[0,0,-1,0],[9E+09,9E+09,9E+09,9E+09,9E+09,9E+09]];
    CONST robtarget T898:=[[33.249920,43.798338,7.749661],[1.000000,0.000000,0.000000,0.000000],[0,0,-1,0],[9E+09,9E+09,9E+09,9E+09,9E+09,9E+09]];
    CONST robtarget T899:=[[33.249920,60.838553,7.749661],[1.000000,0.000000,0.000000,0.000000],[0,0,-1,0],[9E+09,9E+09,9E+09,9E+09,9E+09,9E+09]];
    CONST robtarget T900:=[[31.749914,56.666312,7.749661],[1.000000,0.000000,0.000000,0.000000],[0,0,-1,0],[9E+09,9E+09,9E+09,9E+09,9E+09,9E+09]];
    CONST robtarget T901:=[[31.749914,47.245246,7.749661],[1.000000,0.000000,0.000000,0.000000],[0,0,-1,0],[9E+09,9E+09,9E+09,9E+09,9E+09,9E+09]];
    CONST robtarget T902:=[[30.999911,48.539182,8.249671],[1.000000,0.000000,0.000000,0.000000],[0,0,-1,0],[9E+09,9E+09,9E+09,9E+09,9E+09,9E+09]];
    CONST robtarget T903:=[[30.999911,54.894033,8.249671],[1.000000,0.000000,0.000000,0.000000],[0,0,-1,0],[9E+09,9E+09,9E+09,9E+09,9E+09,9E+09]];
    CONST robtarget T904:=[[30.999911,48.539182,8.249671],[1.000000,0.000000,0.000000,0.000000],[0,0,-1,0],[9E+09,9E+09,9E+09,9E+09,9E+09,9E+09]];
    CONST robtarget T905:=[[30.999911,54.894033,8.249671],[1.000000,0.000000,0.000000,0.000000],[0,0,-1,0],[9E+09,9E+09,9E+09,9E+09,9E+09,9E+09]];
    CONST robtarget T906:=[[32.499917,59.939124,8.249671],[1.000000,0.000000,0.000000,0.000000],[0,0,-1,0],[9E+09,9E+09,9E+09,9E+09,9E+09,9E+09]];
    CONST robtarget T907:=[[32.499917,44.812290,8.249671],[1.000000,0.000000,0.000000,0.000000],[0,0,-1,0],[9E+09,9E+09,9E+09,9E+09,9E+09,9E+09]];
    CONST robtarget T908:=[[33.999923,42.468486,8.249671],[1.000000,0.000000,0.000000,0.000000],[0,0,-1,0],[9E+09,9E+09,9E+09,9E+09,9E+09,9E+09]];
    CONST robtarget T909:=[[33.999923,63.415076,8.249671],[1.000000,0.000000,0.000000,0.000000],[0,0,-1,0],[9E+09,9E+09,9E+09,9E+09,9E+09,9E+09]];
    CONST robtarget T910:=[[35.499929,65.405881,8.249671],[1.000000,0.000000,0.000000,0.000000],[0,0,-1,0],[9E+09,9E+09,9E+09,9E+09,9E+09,9E+09]];
    CONST robtarget T911:=[[35.499929,40.683506,8.249671],[1.000000,0.000000,0.000000,0.000000],[0,0,-1,0],[9E+09,9E+09,9E+09,9E+09,9E+09,9E+09]];
    CONST robtarget T912:=[[36.999935,39.354465,8.249671],[1.000000,0.000000,0.000000,0.000000],[0,0,-1,0],[9E+09,9E+09,9E+09,9E+09,9E+09,9E+09]];
    CONST robtarget T913:=[[36.999935,67.690825,8.249671],[1.000000,0.000000,0.000000,0.000000],[0,0,-1,0],[9E+09,9E+09,9E+09,9E+09,9E+09,9E+09]];
    CONST robtarget T914:=[[38.499941,69.720928,8.249671],[1.000000,0.000000,0.000000,0.000000],[0,0,-1,0],[9E+09,9E+09,9E+09,9E+09,9E+09,9E+09]];
    CONST robtarget T915:=[[38.499941,38.089853,8.249671],[1.000000,0.000000,0.000000,0.000000],[0,0,-1,0],[9E+09,9E+09,9E+09,9E+09,9E+09,9E+09]];
    CONST robtarget T916:=[[39.999947,37.150608,8.249671],[1.000000,0.000000,0.000000,0.000000],[0,0,-1,0],[9E+09,9E+09,9E+09,9E+09,9E+09,9E+09]];
    CONST robtarget T917:=[[39.999947,71.759571,8.249671],[1.000000,0.000000,0.000000,0.000000],[0,0,-1,0],[9E+09,9E+09,9E+09,9E+09,9E+09,9E+09]];
    CONST robtarget T918:=[[41.499953,73.410890,8.249671],[1.000000,0.000000,0.000000,0.000000],[0,0,-1,0],[9E+09,9E+09,9E+09,9E+09,9E+09,9E+09]];
    CONST robtarget T919:=[[41.499953,36.252426,8.249671],[1.000000,0.000000,0.000000,0.000000],[0,0,-1,0],[9E+09,9E+09,9E+09,9E+09,9E+09,9E+09]];
    CONST robtarget T920:=[[42.999959,35.636728,8.249671],[1.000000,0.000000,0.000000,0.000000],[0,0,-1,0],[9E+09,9E+09,9E+09,9E+09,9E+09,9E+09]];
    CONST robtarget T921:=[[42.999959,74.628117,8.249671],[1.000000,0.000000,0.000000,0.000000],[0,0,-1,0],[9E+09,9E+09,9E+09,9E+09,9E+09,9E+09]];
    CONST robtarget T922:=[[44.499965,75.614412,8.249671],[1.000000,0.000000,0.000000,0.000000],[0,0,-1,0],[9E+09,9E+09,9E+09,9E+09,9E+09,9E+09]];
    CONST robtarget T923:=[[44.499965,35.060809,8.249671],[1.000000,0.000000,0.000000,0.000000],[0,0,-1,0],[9E+09,9E+09,9E+09,9E+09,9E+09,9E+09]];
    CONST robtarget T924:=[[45.999971,34.730335,8.249671],[1.000000,0.000000,0.000000,0.000000],[0,0,-1,0],[9E+09,9E+09,9E+09,9E+09,9E+09,9E+09]];
    CONST robtarget T925:=[[45.999971,76.397362,8.249671],[1.000000,0.000000,0.000000,0.000000],[0,0,-1,0],[9E+09,9E+09,9E+09,9E+09,9E+09,9E+09]];
    CONST robtarget T926:=[[47.499977,76.970064,8.249671],[1.000000,0.000000,0.000000,0.000000],[0,0,-1,0],[9E+09,9E+09,9E+09,9E+09,9E+09,9E+09]];
    CONST robtarget T927:=[[47.499977,34.432990,8.249671],[1.000000,0.000000,0.000000,0.000000],[0,0,-1,0],[9E+09,9E+09,9E+09,9E+09,9E+09,9E+09]];
    CONST robtarget T928:=[[48.999983,34.280988,8.249671],[1.000000,0.000000,0.000000,0.000000],[0,0,-1,0],[9E+09,9E+09,9E+09,9E+09,9E+09,9E+09]];
    CONST robtarget T929:=[[48.999983,77.217959,8.249671],[1.000000,0.000000,0.000000,0.000000],[0,0,-1,0],[9E+09,9E+09,9E+09,9E+09,9E+09,9E+09]];
    CONST robtarget T930:=[[50.499989,77.435891,8.249671],[1.000000,0.000000,0.000000,0.000000],[0,0,-1,0],[9E+09,9E+09,9E+09,9E+09,9E+09,9E+09]];
    CONST robtarget T931:=[[50.499989,34.149453,8.249671],[1.000000,0.000000,0.000000,0.000000],[0,0,-1,0],[9E+09,9E+09,9E+09,9E+09,9E+09,9E+09]];
    CONST robtarget T932:=[[51.999995,34.086031,8.249671],[1.000000,0.000000,0.000000,0.000000],[0,0,-1,0],[9E+09,9E+09,9E+09,9E+09,9E+09,9E+09]];
    CONST robtarget T933:=[[51.999995,77.579861,8.249671],[1.000000,0.000000,0.000000,0.000000],[0,0,-1,0],[9E+09,9E+09,9E+09,9E+09,9E+09,9E+09]];
    CONST robtarget T934:=[[53.500001,77.764657,8.249671],[1.000000,0.000000,0.000000,0.000000],[0,0,-1,0],[9E+09,9E+09,9E+09,9E+09,9E+09,9E+09]];
    CONST robtarget T935:=[[53.500001,34.051386,8.249671],[1.000000,0.000000,0.000000,0.000000],[0,0,-1,0],[9E+09,9E+09,9E+09,9E+09,9E+09,9E+09]];
    CONST robtarget T936:=[[55.000007,34.053221,8.249671],[1.000000,0.000000,0.000000,0.000000],[0,0,-1,0],[9E+09,9E+09,9E+09,9E+09,9E+09,9E+09]];
    CONST robtarget T937:=[[55.000007,77.900619,8.249671],[1.000000,0.000000,0.000000,0.000000],[0,0,-1,0],[9E+09,9E+09,9E+09,9E+09,9E+09,9E+09]];
    CONST robtarget T938:=[[56.500013,77.764657,8.249671],[1.000000,0.000000,0.000000,0.000000],[0,0,-1,0],[9E+09,9E+09,9E+09,9E+09,9E+09,9E+09]];
    CONST robtarget T939:=[[56.500013,34.051386,8.249671],[1.000000,0.000000,0.000000,0.000000],[0,0,-1,0],[9E+09,9E+09,9E+09,9E+09,9E+09,9E+09]];
    CONST robtarget T940:=[[58.000019,34.086031,8.249671],[1.000000,0.000000,0.000000,0.000000],[0,0,-1,0],[9E+09,9E+09,9E+09,9E+09,9E+09,9E+09]];
    CONST robtarget T941:=[[58.000019,77.579861,8.249671],[1.000000,0.000000,0.000000,0.000000],[0,0,-1,0],[9E+09,9E+09,9E+09,9E+09,9E+09,9E+09]];
    CONST robtarget T942:=[[59.500025,77.435891,8.249671],[1.000000,0.000000,0.000000,0.000000],[0,0,-1,0],[9E+09,9E+09,9E+09,9E+09,9E+09,9E+09]];
    CONST robtarget T943:=[[59.500025,34.149453,8.249671],[1.000000,0.000000,0.000000,0.000000],[0,0,-1,0],[9E+09,9E+09,9E+09,9E+09,9E+09,9E+09]];
    CONST robtarget T944:=[[61.000031,34.280988,8.249671],[1.000000,0.000000,0.000000,0.000000],[0,0,-1,0],[9E+09,9E+09,9E+09,9E+09,9E+09,9E+09]];
    CONST robtarget T945:=[[61.000031,77.217959,8.249671],[1.000000,0.000000,0.000000,0.000000],[0,0,-1,0],[9E+09,9E+09,9E+09,9E+09,9E+09,9E+09]];
    CONST robtarget T946:=[[62.500037,76.970064,8.249671],[1.000000,0.000000,0.000000,0.000000],[0,0,-1,0],[9E+09,9E+09,9E+09,9E+09,9E+09,9E+09]];
    CONST robtarget T947:=[[62.500037,34.432990,8.249671],[1.000000,0.000000,0.000000,0.000000],[0,0,-1,0],[9E+09,9E+09,9E+09,9E+09,9E+09,9E+09]];
    CONST robtarget T948:=[[64.000043,34.730335,8.249671],[1.000000,0.000000,0.000000,0.000000],[0,0,-1,0],[9E+09,9E+09,9E+09,9E+09,9E+09,9E+09]];
    CONST robtarget T949:=[[64.000043,76.397362,8.249671],[1.000000,0.000000,0.000000,0.000000],[0,0,-1,0],[9E+09,9E+09,9E+09,9E+09,9E+09,9E+09]];
    CONST robtarget T950:=[[65.500049,75.614412,8.249671],[1.000000,0.000000,0.000000,0.000000],[0,0,-1,0],[9E+09,9E+09,9E+09,9E+09,9E+09,9E+09]];
    CONST robtarget T951:=[[65.500049,35.060807,8.249671],[1.000000,0.000000,0.000000,0.000000],[0,0,-1,0],[9E+09,9E+09,9E+09,9E+09,9E+09,9E+09]];
    CONST robtarget T952:=[[67.000055,35.636726,8.249671],[1.000000,0.000000,0.000000,0.000000],[0,0,-1,0],[9E+09,9E+09,9E+09,9E+09,9E+09,9E+09]];
    CONST robtarget T953:=[[67.000055,74.628117,8.249671],[1.000000,0.000000,0.000000,0.000000],[0,0,-1,0],[9E+09,9E+09,9E+09,9E+09,9E+09,9E+09]];
    CONST robtarget T954:=[[68.500061,73.410890,8.249671],[1.000000,0.000000,0.000000,0.000000],[0,0,-1,0],[9E+09,9E+09,9E+09,9E+09,9E+09,9E+09]];
    CONST robtarget T955:=[[68.500061,36.252427,8.249671],[1.000000,0.000000,0.000000,0.000000],[0,0,-1,0],[9E+09,9E+09,9E+09,9E+09,9E+09,9E+09]];
    CONST robtarget T956:=[[70.000067,37.150605,8.249671],[1.000000,0.000000,0.000000,0.000000],[0,0,-1,0],[9E+09,9E+09,9E+09,9E+09,9E+09,9E+09]];
    CONST robtarget T957:=[[70.000067,71.759571,8.249671],[1.000000,0.000000,0.000000,0.000000],[0,0,-1,0],[9E+09,9E+09,9E+09,9E+09,9E+09,9E+09]];
    CONST robtarget T958:=[[71.500073,69.720925,8.249671],[1.000000,0.000000,0.000000,0.000000],[0,0,-1,0],[9E+09,9E+09,9E+09,9E+09,9E+09,9E+09]];
    CONST robtarget T959:=[[71.500073,38.089844,8.249671],[1.000000,0.000000,0.000000,0.000000],[0,0,-1,0],[9E+09,9E+09,9E+09,9E+09,9E+09,9E+09]];
    CONST robtarget T960:=[[73.000079,39.354459,8.249671],[1.000000,0.000000,0.000000,0.000000],[0,0,-1,0],[9E+09,9E+09,9E+09,9E+09,9E+09,9E+09]];
    CONST robtarget T961:=[[73.000079,67.689994,8.249671],[1.000000,0.000000,0.000000,0.000000],[0,0,-1,0],[9E+09,9E+09,9E+09,9E+09,9E+09,9E+09]];
    CONST robtarget T962:=[[74.500085,65.402141,8.249671],[1.000000,0.000000,0.000000,0.000000],[0,0,-1,0],[9E+09,9E+09,9E+09,9E+09,9E+09,9E+09]];
    CONST robtarget T963:=[[74.500085,40.683507,8.249671],[1.000000,0.000000,0.000000,0.000000],[0,0,-1,0],[9E+09,9E+09,9E+09,9E+09,9E+09,9E+09]];
    CONST robtarget T964:=[[76.000091,42.468487,8.249671],[1.000000,0.000000,0.000000,0.000000],[0,0,-1,0],[9E+09,9E+09,9E+09,9E+09,9E+09,9E+09]];
    CONST robtarget T965:=[[76.000091,63.413684,8.249671],[1.000000,0.000000,0.000000,0.000000],[0,0,-1,0],[9E+09,9E+09,9E+09,9E+09,9E+09,9E+09]];
    CONST robtarget T966:=[[77.500097,59.934842,8.249671],[1.000000,0.000000,0.000000,0.000000],[0,0,-1,0],[9E+09,9E+09,9E+09,9E+09,9E+09,9E+09]];
    CONST robtarget T967:=[[77.500097,44.812292,8.249671],[1.000000,0.000000,0.000000,0.000000],[0,0,-1,0],[9E+09,9E+09,9E+09,9E+09,9E+09,9E+09]];
    CONST robtarget T968:=[[79.000103,48.539185,8.249671],[1.000000,0.000000,0.000000,0.000000],[0,0,-1,0],[9E+09,9E+09,9E+09,9E+09,9E+09,9E+09]];
    CONST robtarget T969:=[[79.000103,54.893679,8.249671],[1.000000,0.000000,0.000000,0.000000],[0,0,-1,0],[9E+09,9E+09,9E+09,9E+09,9E+09,9E+09]];
    CONST robtarget T970:=[[79.000103,48.138084,8.749681],[1.000000,0.000000,0.000000,0.000000],[0,0,-1,0],[9E+09,9E+09,9E+09,9E+09,9E+09,9E+09]];
    CONST robtarget T971:=[[79.000103,56.010647,8.749681],[1.000000,0.000000,0.000000,0.000000],[0,0,-1,0],[9E+09,9E+09,9E+09,9E+09,9E+09,9E+09]];
    CONST robtarget T972:=[[79.000103,48.138084,8.749681],[1.000000,0.000000,0.000000,0.000000],[0,0,-1,0],[9E+09,9E+09,9E+09,9E+09,9E+09,9E+09]];
    CONST robtarget T973:=[[79.000103,56.010647,8.749681],[1.000000,0.000000,0.000000,0.000000],[0,0,-1,0],[9E+09,9E+09,9E+09,9E+09,9E+09,9E+09]];
    CONST robtarget T974:=[[77.500097,60.733005,8.749681],[1.000000,0.000000,0.000000,0.000000],[0,0,-1,0],[9E+09,9E+09,9E+09,9E+09,9E+09,9E+09]];
    CONST robtarget T975:=[[77.500097,44.419564,8.749681],[1.000000,0.000000,0.000000,0.000000],[0,0,-1,0],[9E+09,9E+09,9E+09,9E+09,9E+09,9E+09]];
    CONST robtarget T976:=[[76.000091,42.174834,8.749681],[1.000000,0.000000,0.000000,0.000000],[0,0,-1,0],[9E+09,9E+09,9E+09,9E+09,9E+09,9E+09]];
    CONST robtarget T977:=[[76.000091,64.251287,8.749681],[1.000000,0.000000,0.000000,0.000000],[0,0,-1,0],[9E+09,9E+09,9E+09,9E+09,9E+09,9E+09]];
    CONST robtarget T978:=[[74.500085,65.965142,8.749681],[1.000000,0.000000,0.000000,0.000000],[0,0,-1,0],[9E+09,9E+09,9E+09,9E+09,9E+09,9E+09]];
    CONST robtarget T979:=[[74.500085,40.369776,8.749681],[1.000000,0.000000,0.000000,0.000000],[0,0,-1,0],[9E+09,9E+09,9E+09,9E+09,9E+09,9E+09]];
    CONST robtarget T980:=[[73.000079,39.031854,8.749681],[1.000000,0.000000,0.000000,0.000000],[0,0,-1,0],[9E+09,9E+09,9E+09,9E+09,9E+09,9E+09]];
    CONST robtarget T981:=[[73.000079,67.883091,8.749681],[1.000000,0.000000,0.000000,0.000000],[0,0,-1,0],[9E+09,9E+09,9E+09,9E+09,9E+09,9E+09]];
    CONST robtarget T982:=[[71.500073,69.943893,8.749681],[1.000000,0.000000,0.000000,0.000000],[0,0,-1,0],[9E+09,9E+09,9E+09,9E+09,9E+09,9E+09]];
    CONST robtarget T983:=[[71.500073,37.797738,8.749681],[1.000000,0.000000,0.000000,0.000000],[0,0,-1,0],[9E+09,9E+09,9E+09,9E+09,9E+09,9E+09]];
    CONST robtarget T984:=[[70.000067,36.858498,8.749681],[1.000000,0.000000,0.000000,0.000000],[0,0,-1,0],[9E+09,9E+09,9E+09,9E+09,9E+09,9E+09]];
    CONST robtarget T985:=[[70.000067,71.982539,8.749681],[1.000000,0.000000,0.000000,0.000000],[0,0,-1,0],[9E+09,9E+09,9E+09,9E+09,9E+09,9E+09]];
    CONST robtarget T986:=[[68.500061,73.658846,8.749681],[1.000000,0.000000,0.000000,0.000000],[0,0,-1,0],[9E+09,9E+09,9E+09,9E+09,9E+09,9E+09]];
    CONST robtarget T987:=[[68.500061,35.980011,8.749681],[1.000000,0.000000,0.000000,0.000000],[0,0,-1,0],[9E+09,9E+09,9E+09,9E+09,9E+09,9E+09]];
    CONST robtarget T988:=[[67.000055,35.364572,8.749681],[1.000000,0.000000,0.000000,0.000000],[0,0,-1,0],[9E+09,9E+09,9E+09,9E+09,9E+09,9E+09]];
    CONST robtarget T989:=[[67.000055,74.909593,8.749681],[1.000000,0.000000,0.000000,0.000000],[0,0,-1,0],[9E+09,9E+09,9E+09,9E+09,9E+09,9E+09]];
    CONST robtarget T990:=[[65.500049,75.874338,8.749681],[1.000000,0.000000,0.000000,0.000000],[0,0,-1,0],[9E+09,9E+09,9E+09,9E+09,9E+09,9E+09]];
    CONST robtarget T991:=[[65.500049,34.793548,8.749681],[1.000000,0.000000,0.000000,0.000000],[0,0,-1,0],[9E+09,9E+09,9E+09,9E+09,9E+09,9E+09]];
    CONST robtarget T992:=[[64.000043,34.463155,8.749681],[1.000000,0.000000,0.000000,0.000000],[0,0,-1,0],[9E+09,9E+09,9E+09,9E+09,9E+09,9E+09]];
    CONST robtarget T993:=[[64.000043,76.593588,8.749681],[1.000000,0.000000,0.000000,0.000000],[0,0,-1,0],[9E+09,9E+09,9E+09,9E+09,9E+09,9E+09]];
    CONST robtarget T994:=[[62.500037,77.118599,8.749681],[1.000000,0.000000,0.000000,0.000000],[0,0,-1,0],[9E+09,9E+09,9E+09,9E+09,9E+09,9E+09]];
    CONST robtarget T995:=[[62.500037,34.169157,8.749681],[1.000000,0.000000,0.000000,0.000000],[0,0,-1,0],[9E+09,9E+09,9E+09,9E+09,9E+09,9E+09]];
    CONST robtarget T996:=[[61.000031,34.021518,8.749681],[1.000000,0.000000,0.000000,0.000000],[0,0,-1,0],[9E+09,9E+09,9E+09,9E+09,9E+09,9E+09]];
    CONST robtarget T997:=[[61.000031,77.382156,8.749681],[1.000000,0.000000,0.000000,0.000000],[0,0,-1,0],[9E+09,9E+09,9E+09,9E+09,9E+09,9E+09]];
    CONST robtarget T998:=[[59.500025,77.621042,8.749681],[1.000000,0.000000,0.000000,0.000000],[0,0,-1,0],[9E+09,9E+09,9E+09,9E+09,9E+09,9E+09]];
    CONST robtarget T999:=[[59.500025,33.889766,8.749681],[1.000000,0.000000,0.000000,0.000000],[0,0,-1,0],[9E+09,9E+09,9E+09,9E+09,9E+09,9E+09]];
    CONST robtarget T1000:=[[58.000019,33.824081,8.749681],[1.000000,0.000000,0.000000,0.000000],[0,0,-1,0],[9E+09,9E+09,9E+09,9E+09,9E+09,9E+09]];
    CONST robtarget T1001:=[[58.000019,77.765012,8.749681],[1.000000,0.000000,0.000000,0.000000],[0,0,-1,0],[9E+09,9E+09,9E+09,9E+09,9E+09,9E+09]];
    CONST robtarget T1002:=[[56.500013,77.949722,8.749681],[1.000000,0.000000,0.000000,0.000000],[0,0,-1,0],[9E+09,9E+09,9E+09,9E+09,9E+09,9E+09]];
    CONST robtarget T1003:=[[56.500013,33.786351,8.749681],[1.000000,0.000000,0.000000,0.000000],[0,0,-1,0],[9E+09,9E+09,9E+09,9E+09,9E+09,9E+09]];
    CONST robtarget T1004:=[[55.000007,33.787413,8.749681],[1.000000,0.000000,0.000000,0.000000],[0,0,-1,0],[9E+09,9E+09,9E+09,9E+09,9E+09,9E+09]];
    CONST robtarget T1005:=[[55.000007,78.097383,8.749681],[1.000000,0.000000,0.000000,0.000000],[0,0,-1,0],[9E+09,9E+09,9E+09,9E+09,9E+09,9E+09]];
    CONST robtarget T1006:=[[53.500001,77.949722,8.749681],[1.000000,0.000000,0.000000,0.000000],[0,0,-1,0],[9E+09,9E+09,9E+09,9E+09,9E+09,9E+09]];
    CONST robtarget T1007:=[[53.500001,33.786351,8.749681],[1.000000,0.000000,0.000000,0.000000],[0,0,-1,0],[9E+09,9E+09,9E+09,9E+09,9E+09,9E+09]];
    CONST robtarget T1008:=[[51.999995,33.824082,8.749681],[1.000000,0.000000,0.000000,0.000000],[0,0,-1,0],[9E+09,9E+09,9E+09,9E+09,9E+09,9E+09]];
    CONST robtarget T1009:=[[51.999995,77.765012,8.749681],[1.000000,0.000000,0.000000,0.000000],[0,0,-1,0],[9E+09,9E+09,9E+09,9E+09,9E+09,9E+09]];
    CONST robtarget T1010:=[[50.499989,77.621042,8.749681],[1.000000,0.000000,0.000000,0.000000],[0,0,-1,0],[9E+09,9E+09,9E+09,9E+09,9E+09,9E+09]];
    CONST robtarget T1011:=[[50.499989,33.889766,8.749681],[1.000000,0.000000,0.000000,0.000000],[0,0,-1,0],[9E+09,9E+09,9E+09,9E+09,9E+09,9E+09]];
    CONST robtarget T1012:=[[48.999983,34.021518,8.749681],[1.000000,0.000000,0.000000,0.000000],[0,0,-1,0],[9E+09,9E+09,9E+09,9E+09,9E+09,9E+09]];
    CONST robtarget T1013:=[[48.999983,77.382156,8.749681],[1.000000,0.000000,0.000000,0.000000],[0,0,-1,0],[9E+09,9E+09,9E+09,9E+09,9E+09,9E+09]];
    CONST robtarget T1014:=[[47.499977,77.118599,8.749681],[1.000000,0.000000,0.000000,0.000000],[0,0,-1,0],[9E+09,9E+09,9E+09,9E+09,9E+09,9E+09]];
    CONST robtarget T1015:=[[47.499977,34.169157,8.749681],[1.000000,0.000000,0.000000,0.000000],[0,0,-1,0],[9E+09,9E+09,9E+09,9E+09,9E+09,9E+09]];
    CONST robtarget T1016:=[[45.999971,34.463156,8.749681],[1.000000,0.000000,0.000000,0.000000],[0,0,-1,0],[9E+09,9E+09,9E+09,9E+09,9E+09,9E+09]];
    CONST robtarget T1017:=[[45.999971,76.593588,8.749681],[1.000000,0.000000,0.000000,0.000000],[0,0,-1,0],[9E+09,9E+09,9E+09,9E+09,9E+09,9E+09]];
    CONST robtarget T1018:=[[44.499965,75.874338,8.749681],[1.000000,0.000000,0.000000,0.000000],[0,0,-1,0],[9E+09,9E+09,9E+09,9E+09,9E+09,9E+09]];
    CONST robtarget T1019:=[[44.499965,34.793550,8.749681],[1.000000,0.000000,0.000000,0.000000],[0,0,-1,0],[9E+09,9E+09,9E+09,9E+09,9E+09,9E+09]];
    CONST robtarget T1020:=[[42.999959,35.364573,8.749681],[1.000000,0.000000,0.000000,0.000000],[0,0,-1,0],[9E+09,9E+09,9E+09,9E+09,9E+09,9E+09]];
    CONST robtarget T1021:=[[42.999959,74.909593,8.749681],[1.000000,0.000000,0.000000,0.000000],[0,0,-1,0],[9E+09,9E+09,9E+09,9E+09,9E+09,9E+09]];
    CONST robtarget T1022:=[[41.499953,73.658845,8.749681],[1.000000,0.000000,0.000000,0.000000],[0,0,-1,0],[9E+09,9E+09,9E+09,9E+09,9E+09,9E+09]];
    CONST robtarget T1023:=[[41.499953,35.980008,8.749681],[1.000000,0.000000,0.000000,0.000000],[0,0,-1,0],[9E+09,9E+09,9E+09,9E+09,9E+09,9E+09]];
    CONST robtarget T1024:=[[39.999947,36.858499,8.749681],[1.000000,0.000000,0.000000,0.000000],[0,0,-1,0],[9E+09,9E+09,9E+09,9E+09,9E+09,9E+09]];
    CONST robtarget T1025:=[[39.999947,71.982538,8.749681],[1.000000,0.000000,0.000000,0.000000],[0,0,-1,0],[9E+09,9E+09,9E+09,9E+09,9E+09,9E+09]];
    CONST robtarget T1026:=[[38.499941,69.943895,8.749681],[1.000000,0.000000,0.000000,0.000000],[0,0,-1,0],[9E+09,9E+09,9E+09,9E+09,9E+09,9E+09]];
    CONST robtarget T1027:=[[38.499941,37.797744,8.749681],[1.000000,0.000000,0.000000,0.000000],[0,0,-1,0],[9E+09,9E+09,9E+09,9E+09,9E+09,9E+09]];
    CONST robtarget T1028:=[[36.999935,39.031857,8.749681],[1.000000,0.000000,0.000000,0.000000],[0,0,-1,0],[9E+09,9E+09,9E+09,9E+09,9E+09,9E+09]];
    CONST robtarget T1029:=[[36.999935,67.883509,8.749681],[1.000000,0.000000,0.000000,0.000000],[0,0,-1,0],[9E+09,9E+09,9E+09,9E+09,9E+09,9E+09]];
    CONST robtarget T1030:=[[35.499929,65.964613,8.749681],[1.000000,0.000000,0.000000,0.000000],[0,0,-1,0],[9E+09,9E+09,9E+09,9E+09,9E+09,9E+09]];
    CONST robtarget T1031:=[[35.499929,40.369775,8.749681],[1.000000,0.000000,0.000000,0.000000],[0,0,-1,0],[9E+09,9E+09,9E+09,9E+09,9E+09,9E+09]];
    CONST robtarget T1032:=[[33.999923,42.174834,8.749681],[1.000000,0.000000,0.000000,0.000000],[0,0,-1,0],[9E+09,9E+09,9E+09,9E+09,9E+09,9E+09]];
    CONST robtarget T1033:=[[33.999923,64.251756,8.749681],[1.000000,0.000000,0.000000,0.000000],[0,0,-1,0],[9E+09,9E+09,9E+09,9E+09,9E+09,9E+09]];
    CONST robtarget T1034:=[[32.499917,60.735092,8.749681],[1.000000,0.000000,0.000000,0.000000],[0,0,-1,0],[9E+09,9E+09,9E+09,9E+09,9E+09,9E+09]];
    CONST robtarget T1035:=[[32.499917,44.419563,8.749681],[1.000000,0.000000,0.000000,0.000000],[0,0,-1,0],[9E+09,9E+09,9E+09,9E+09,9E+09,9E+09]];
    CONST robtarget T1036:=[[30.999911,48.138083,8.749681],[1.000000,0.000000,0.000000,0.000000],[0,0,-1,0],[9E+09,9E+09,9E+09,9E+09,9E+09,9E+09]];
    CONST robtarget T1037:=[[30.999911,56.009549,8.749681],[1.000000,0.000000,0.000000,0.000000],[0,0,-1,0],[9E+09,9E+09,9E+09,9E+09,9E+09,9E+09]];
    CONST robtarget T1038:=[[30.999911,47.736983,9.249691],[1.000000,0.000000,0.000000,0.000000],[0,0,-1,0],[9E+09,9E+09,9E+09,9E+09,9E+09,9E+09]];
    CONST robtarget T1039:=[[30.999911,56.494030,9.249691],[1.000000,0.000000,0.000000,0.000000],[0,0,-1,0],[9E+09,9E+09,9E+09,9E+09,9E+09,9E+09]];
    CONST robtarget T1040:=[[30.999911,47.736983,9.249691],[1.000000,0.000000,0.000000,0.000000],[0,0,-1,0],[9E+09,9E+09,9E+09,9E+09,9E+09,9E+09]];
    CONST robtarget T1041:=[[30.999911,56.494030,9.249691],[1.000000,0.000000,0.000000,0.000000],[0,0,-1,0],[9E+09,9E+09,9E+09,9E+09,9E+09,9E+09]];
    CONST robtarget T1042:=[[32.499917,61.480186,9.249691],[1.000000,0.000000,0.000000,0.000000],[0,0,-1,0],[9E+09,9E+09,9E+09,9E+09,9E+09,9E+09]];
    CONST robtarget T1043:=[[32.499917,44.026837,9.249691],[1.000000,0.000000,0.000000,0.000000],[0,0,-1,0],[9E+09,9E+09,9E+09,9E+09,9E+09,9E+09]];
    CONST robtarget T1044:=[[33.999923,41.881181,9.249691],[1.000000,0.000000,0.000000,0.000000],[0,0,-1,0],[9E+09,9E+09,9E+09,9E+09,9E+09,9E+09]];
    CONST robtarget T1045:=[[33.999923,64.997798,9.249691],[1.000000,0.000000,0.000000,0.000000],[0,0,-1,0],[9E+09,9E+09,9E+09,9E+09,9E+09,9E+09]];
    CONST robtarget T1046:=[[35.499929,66.314453,9.249691],[1.000000,0.000000,0.000000,0.000000],[0,0,-1,0],[9E+09,9E+09,9E+09,9E+09,9E+09,9E+09]];
    CONST robtarget T1047:=[[35.499929,40.069821,9.249691],[1.000000,0.000000,0.000000,0.000000],[0,0,-1,0],[9E+09,9E+09,9E+09,9E+09,9E+09,9E+09]];
    CONST robtarget T1048:=[[36.999935,38.709250,9.249691],[1.000000,0.000000,0.000000,0.000000],[0,0,-1,0],[9E+09,9E+09,9E+09,9E+09,9E+09,9E+09]];
    CONST robtarget T1049:=[[36.999935,67.899472,9.249691],[1.000000,0.000000,0.000000,0.000000],[0,0,-1,0],[9E+09,9E+09,9E+09,9E+09,9E+09,9E+09]];
    CONST robtarget T1050:=[[38.499941,70.030654,9.249691],[1.000000,0.000000,0.000000,0.000000],[0,0,-1,0],[9E+09,9E+09,9E+09,9E+09,9E+09,9E+09]];
    CONST robtarget T1051:=[[38.499941,37.505635,9.249691],[1.000000,0.000000,0.000000,0.000000],[0,0,-1,0],[9E+09,9E+09,9E+09,9E+09,9E+09,9E+09]];
    CONST robtarget T1052:=[[39.999947,36.569003,9.249691],[1.000000,0.000000,0.000000,0.000000],[0,0,-1,0],[9E+09,9E+09,9E+09,9E+09,9E+09,9E+09]];
    CONST robtarget T1053:=[[39.999947,72.074712,9.249691],[1.000000,0.000000,0.000000,0.000000],[0,0,-1,0],[9E+09,9E+09,9E+09,9E+09,9E+09,9E+09]];
    CONST robtarget T1054:=[[41.499953,73.774999,9.249691],[1.000000,0.000000,0.000000,0.000000],[0,0,-1,0],[9E+09,9E+09,9E+09,9E+09,9E+09,9E+09]];
    CONST robtarget T1055:=[[41.499953,35.707590,9.249691],[1.000000,0.000000,0.000000,0.000000],[0,0,-1,0],[9E+09,9E+09,9E+09,9E+09,9E+09,9E+09]];
    CONST robtarget T1056:=[[42.999959,35.092418,9.249691],[1.000000,0.000000,0.000000,0.000000],[0,0,-1,0],[9E+09,9E+09,9E+09,9E+09,9E+09,9E+09]];
    CONST robtarget T1057:=[[42.999959,75.059747,9.249691],[1.000000,0.000000,0.000000,0.000000],[0,0,-1,0],[9E+09,9E+09,9E+09,9E+09,9E+09,9E+09]];
    CONST robtarget T1058:=[[44.499965,76.018003,9.249691],[1.000000,0.000000,0.000000,0.000000],[0,0,-1,0],[9E+09,9E+09,9E+09,9E+09,9E+09,9E+09]];
    CONST robtarget T1059:=[[44.499965,34.526291,9.249691],[1.000000,0.000000,0.000000,0.000000],[0,0,-1,0],[9E+09,9E+09,9E+09,9E+09,9E+09,9E+09]];
    CONST robtarget T1060:=[[45.999971,34.199542,9.249691],[1.000000,0.000000,0.000000,0.000000],[0,0,-1,0],[9E+09,9E+09,9E+09,9E+09,9E+09,9E+09]];
    CONST robtarget T1061:=[[45.999971,76.742135,9.249691],[1.000000,0.000000,0.000000,0.000000],[0,0,-1,0],[9E+09,9E+09,9E+09,9E+09,9E+09,9E+09]];
    CONST robtarget T1062:=[[47.499977,77.267135,9.249691],[1.000000,0.000000,0.000000,0.000000],[0,0,-1,0],[9E+09,9E+09,9E+09,9E+09,9E+09,9E+09]];
    CONST robtarget T1063:=[[47.499977,33.905324,9.249691],[1.000000,0.000000,0.000000,0.000000],[0,0,-1,0],[9E+09,9E+09,9E+09,9E+09,9E+09,9E+09]];
    CONST robtarget T1064:=[[48.999983,33.762048,9.249691],[1.000000,0.000000,0.000000,0.000000],[0,0,-1,0],[9E+09,9E+09,9E+09,9E+09,9E+09,9E+09]];
    CONST robtarget T1065:=[[48.999983,77.546354,9.249691],[1.000000,0.000000,0.000000,0.000000],[0,0,-1,0],[9E+09,9E+09,9E+09,9E+09,9E+09,9E+09]];
    CONST robtarget T1066:=[[50.499989,77.797778,9.249691],[1.000000,0.000000,0.000000,0.000000],[0,0,-1,0],[9E+09,9E+09,9E+09,9E+09,9E+09,9E+09]];
    CONST robtarget T1067:=[[50.499989,33.630080,9.249691],[1.000000,0.000000,0.000000,0.000000],[0,0,-1,0],[9E+09,9E+09,9E+09,9E+09,9E+09,9E+09]];
    CONST robtarget T1068:=[[51.999995,33.562132,9.249691],[1.000000,0.000000,0.000000,0.000000],[0,0,-1,0],[9E+09,9E+09,9E+09,9E+09,9E+09,9E+09]];
    CONST robtarget T1069:=[[51.999995,77.950162,9.249691],[1.000000,0.000000,0.000000,0.000000],[0,0,-1,0],[9E+09,9E+09,9E+09,9E+09,9E+09,9E+09]];
    CONST robtarget T1070:=[[53.500001,78.142049,9.249691],[1.000000,0.000000,0.000000,0.000000],[0,0,-1,0],[9E+09,9E+09,9E+09,9E+09,9E+09,9E+09]];
    CONST robtarget T1071:=[[53.500001,33.524160,9.249691],[1.000000,0.000000,0.000000,0.000000],[0,0,-1,0],[9E+09,9E+09,9E+09,9E+09,9E+09,9E+09]];
    CONST robtarget T1072:=[[55.000007,33.521604,9.249691],[1.000000,0.000000,0.000000,0.000000],[0,0,-1,0],[9E+09,9E+09,9E+09,9E+09,9E+09,9E+09]];
    CONST robtarget T1073:=[[55.000007,78.294147,9.249691],[1.000000,0.000000,0.000000,0.000000],[0,0,-1,0],[9E+09,9E+09,9E+09,9E+09,9E+09,9E+09]];
    CONST robtarget T1074:=[[56.500013,78.142049,9.249691],[1.000000,0.000000,0.000000,0.000000],[0,0,-1,0],[9E+09,9E+09,9E+09,9E+09,9E+09,9E+09]];
    CONST robtarget T1075:=[[56.500013,33.524159,9.249691],[1.000000,0.000000,0.000000,0.000000],[0,0,-1,0],[9E+09,9E+09,9E+09,9E+09,9E+09,9E+09]];
    CONST robtarget T1076:=[[58.000019,33.562130,9.249691],[1.000000,0.000000,0.000000,0.000000],[0,0,-1,0],[9E+09,9E+09,9E+09,9E+09,9E+09,9E+09]];
    CONST robtarget T1077:=[[58.000019,77.950162,9.249691],[1.000000,0.000000,0.000000,0.000000],[0,0,-1,0],[9E+09,9E+09,9E+09,9E+09,9E+09,9E+09]];
    CONST robtarget T1078:=[[59.500025,77.797778,9.249691],[1.000000,0.000000,0.000000,0.000000],[0,0,-1,0],[9E+09,9E+09,9E+09,9E+09,9E+09,9E+09]];
    CONST robtarget T1079:=[[59.500025,33.630079,9.249691],[1.000000,0.000000,0.000000,0.000000],[0,0,-1,0],[9E+09,9E+09,9E+09,9E+09,9E+09,9E+09]];
    CONST robtarget T1080:=[[61.000031,33.762048,9.249691],[1.000000,0.000000,0.000000,0.000000],[0,0,-1,0],[9E+09,9E+09,9E+09,9E+09,9E+09,9E+09]];
    CONST robtarget T1081:=[[61.000031,77.546354,9.249691],[1.000000,0.000000,0.000000,0.000000],[0,0,-1,0],[9E+09,9E+09,9E+09,9E+09,9E+09,9E+09]];
    CONST robtarget T1082:=[[62.500037,77.267135,9.249691],[1.000000,0.000000,0.000000,0.000000],[0,0,-1,0],[9E+09,9E+09,9E+09,9E+09,9E+09,9E+09]];
    CONST robtarget T1083:=[[62.500037,33.905324,9.249691],[1.000000,0.000000,0.000000,0.000000],[0,0,-1,0],[9E+09,9E+09,9E+09,9E+09,9E+09,9E+09]];
    CONST robtarget T1084:=[[64.000043,34.199542,9.249691],[1.000000,0.000000,0.000000,0.000000],[0,0,-1,0],[9E+09,9E+09,9E+09,9E+09,9E+09,9E+09]];
    CONST robtarget T1085:=[[64.000043,76.742136,9.249691],[1.000000,0.000000,0.000000,0.000000],[0,0,-1,0],[9E+09,9E+09,9E+09,9E+09,9E+09,9E+09]];
    CONST robtarget T1086:=[[65.500049,76.018003,9.249691],[1.000000,0.000000,0.000000,0.000000],[0,0,-1,0],[9E+09,9E+09,9E+09,9E+09,9E+09,9E+09]];
    CONST robtarget T1087:=[[65.500049,34.526290,9.249691],[1.000000,0.000000,0.000000,0.000000],[0,0,-1,0],[9E+09,9E+09,9E+09,9E+09,9E+09,9E+09]];
    CONST robtarget T1088:=[[67.000055,35.092417,9.249691],[1.000000,0.000000,0.000000,0.000000],[0,0,-1,0],[9E+09,9E+09,9E+09,9E+09,9E+09,9E+09]];
    CONST robtarget T1089:=[[67.000055,75.059748,9.249691],[1.000000,0.000000,0.000000,0.000000],[0,0,-1,0],[9E+09,9E+09,9E+09,9E+09,9E+09,9E+09]];
    CONST robtarget T1090:=[[68.500061,73.775000,9.249691],[1.000000,0.000000,0.000000,0.000000],[0,0,-1,0],[9E+09,9E+09,9E+09,9E+09,9E+09,9E+09]];
    CONST robtarget T1091:=[[68.500061,35.707595,9.249691],[1.000000,0.000000,0.000000,0.000000],[0,0,-1,0],[9E+09,9E+09,9E+09,9E+09,9E+09,9E+09]];
    CONST robtarget T1092:=[[70.000067,36.569004,9.249691],[1.000000,0.000000,0.000000,0.000000],[0,0,-1,0],[9E+09,9E+09,9E+09,9E+09,9E+09,9E+09]];
    CONST robtarget T1093:=[[70.000067,72.074713,9.249691],[1.000000,0.000000,0.000000,0.000000],[0,0,-1,0],[9E+09,9E+09,9E+09,9E+09,9E+09,9E+09]];
    CONST robtarget T1094:=[[71.500073,70.030653,9.249691],[1.000000,0.000000,0.000000,0.000000],[0,0,-1,0],[9E+09,9E+09,9E+09,9E+09,9E+09,9E+09]];
    CONST robtarget T1095:=[[71.500073,37.505631,9.249691],[1.000000,0.000000,0.000000,0.000000],[0,0,-1,0],[9E+09,9E+09,9E+09,9E+09,9E+09,9E+09]];
    CONST robtarget T1096:=[[73.000079,38.709248,9.249691],[1.000000,0.000000,0.000000,0.000000],[0,0,-1,0],[9E+09,9E+09,9E+09,9E+09,9E+09,9E+09]];
    CONST robtarget T1097:=[[73.000079,67.899001,9.249691],[1.000000,0.000000,0.000000,0.000000],[0,0,-1,0],[9E+09,9E+09,9E+09,9E+09,9E+09,9E+09]];
    CONST robtarget T1098:=[[74.500085,66.314289,9.249691],[1.000000,0.000000,0.000000,0.000000],[0,0,-1,0],[9E+09,9E+09,9E+09,9E+09,9E+09,9E+09]];
    CONST robtarget T1099:=[[74.500085,40.069821,9.249691],[1.000000,0.000000,0.000000,0.000000],[0,0,-1,0],[9E+09,9E+09,9E+09,9E+09,9E+09,9E+09]];
    CONST robtarget T1100:=[[76.000091,41.881181,9.249691],[1.000000,0.000000,0.000000,0.000000],[0,0,-1,0],[9E+09,9E+09,9E+09,9E+09,9E+09,9E+09]];
    CONST robtarget T1101:=[[76.000091,64.997467,9.249691],[1.000000,0.000000,0.000000,0.000000],[0,0,-1,0],[9E+09,9E+09,9E+09,9E+09,9E+09,9E+09]];
    CONST robtarget T1102:=[[77.500097,61.479959,9.249691],[1.000000,0.000000,0.000000,0.000000],[0,0,-1,0],[9E+09,9E+09,9E+09,9E+09,9E+09,9E+09]];
    CONST robtarget T1103:=[[77.500097,44.026837,9.249691],[1.000000,0.000000,0.000000,0.000000],[0,0,-1,0],[9E+09,9E+09,9E+09,9E+09,9E+09,9E+09]];
    CONST robtarget T1104:=[[79.000103,47.736983,9.249691],[1.000000,0.000000,0.000000,0.000000],[0,0,-1,0],[9E+09,9E+09,9E+09,9E+09,9E+09,9E+09]];
    CONST robtarget T1105:=[[79.000103,56.491285,9.249691],[1.000000,0.000000,0.000000,0.000000],[0,0,-1,0],[9E+09,9E+09,9E+09,9E+09,9E+09,9E+09]];
    CONST robtarget T1106:=[[79.000102,47.335881,9.749701],[1.000000,0.000000,0.000000,0.000000],[0,0,-1,0],[9E+09,9E+09,9E+09,9E+09,9E+09,9E+09]];
    CONST robtarget T1107:=[[79.000102,56.840451,9.749701],[1.000000,0.000000,0.000000,0.000000],[0,0,-1,0],[9E+09,9E+09,9E+09,9E+09,9E+09,9E+09]];
    CONST robtarget T1108:=[[79.000102,47.335881,9.749701],[1.000000,0.000000,0.000000,0.000000],[0,0,-1,0],[9E+09,9E+09,9E+09,9E+09,9E+09,9E+09]];
    CONST robtarget T1109:=[[79.000102,56.840451,9.749701],[1.000000,0.000000,0.000000,0.000000],[0,0,-1,0],[9E+09,9E+09,9E+09,9E+09,9E+09,9E+09]];
    CONST robtarget T1110:=[[77.500096,62.226914,9.749701],[1.000000,0.000000,0.000000,0.000000],[0,0,-1,0],[9E+09,9E+09,9E+09,9E+09,9E+09,9E+09]];
    CONST robtarget T1111:=[[77.500096,43.634109,9.749701],[1.000000,0.000000,0.000000,0.000000],[0,0,-1,0],[9E+09,9E+09,9E+09,9E+09,9E+09,9E+09]];
    CONST robtarget T1112:=[[76.000090,41.553005,9.749701],[1.000000,0.000000,0.000000,0.000000],[0,0,-1,0],[9E+09,9E+09,9E+09,9E+09,9E+09,9E+09]];
    CONST robtarget T1113:=[[76.000090,65.718144,9.749701],[1.000000,0.000000,0.000000,0.000000],[0,0,-1,0],[9E+09,9E+09,9E+09,9E+09,9E+09,9E+09]];
    CONST robtarget T1114:=[[74.500084,66.564609,9.749701],[1.000000,0.000000,0.000000,0.000000],[0,0,-1,0],[9E+09,9E+09,9E+09,9E+09,9E+09,9E+09]];
    CONST robtarget T1115:=[[74.500084,39.769865,9.749701],[1.000000,0.000000,0.000000,0.000000],[0,0,-1,0],[9E+09,9E+09,9E+09,9E+09,9E+09,9E+09]];
    CONST robtarget T1116:=[[73.000078,38.386642,9.749701],[1.000000,0.000000,0.000000,0.000000],[0,0,-1,0],[9E+09,9E+09,9E+09,9E+09,9E+09,9E+09]];
    CONST robtarget T1117:=[[73.000078,67.905875,9.749701],[1.000000,0.000000,0.000000,0.000000],[0,0,-1,0],[9E+09,9E+09,9E+09,9E+09,9E+09,9E+09]];
    CONST robtarget T1118:=[[71.500072,70.071653,9.749701],[1.000000,0.000000,0.000000,0.000000],[0,0,-1,0],[9E+09,9E+09,9E+09,9E+09,9E+09,9E+09]];
    CONST robtarget T1119:=[[71.500072,37.213525,9.749701],[1.000000,0.000000,0.000000,0.000000],[0,0,-1,0],[9E+09,9E+09,9E+09,9E+09,9E+09,9E+09]];
    CONST robtarget T1120:=[[70.000066,36.281329,9.749701],[1.000000,0.000000,0.000000,0.000000],[0,0,-1,0],[9E+09,9E+09,9E+09,9E+09,9E+09,9E+09]];
    CONST robtarget T1121:=[[70.000066,72.149606,9.749701],[1.000000,0.000000,0.000000,0.000000],[0,0,-1,0],[9E+09,9E+09,9E+09,9E+09,9E+09,9E+09]];
    CONST robtarget T1122:=[[68.500060,73.885586,9.749701],[1.000000,0.000000,0.000000,0.000000],[0,0,-1,0],[9E+09,9E+09,9E+09,9E+09,9E+09,9E+09]];
    CONST robtarget T1123:=[[68.500060,35.435178,9.749701],[1.000000,0.000000,0.000000,0.000000],[0,0,-1,0],[9E+09,9E+09,9E+09,9E+09,9E+09,9E+09]];
    CONST robtarget T1124:=[[67.000054,34.820111,9.749701],[1.000000,0.000000,0.000000,0.000000],[0,0,-1,0],[9E+09,9E+09,9E+09,9E+09,9E+09,9E+09]];
    CONST robtarget T1125:=[[67.000054,75.188417,9.749701],[1.000000,0.000000,0.000000,0.000000],[0,0,-1,0],[9E+09,9E+09,9E+09,9E+09,9E+09,9E+09]];
    CONST robtarget T1126:=[[65.500048,76.161668,9.749701],[1.000000,0.000000,0.000000,0.000000],[0,0,-1,0],[9E+09,9E+09,9E+09,9E+09,9E+09,9E+09]];
    CONST robtarget T1127:=[[65.500048,34.259032,9.749701],[1.000000,0.000000,0.000000,0.000000],[0,0,-1,0],[9E+09,9E+09,9E+09,9E+09,9E+09,9E+09]];
    CONST robtarget T1128:=[[64.000042,33.935928,9.749701],[1.000000,0.000000,0.000000,0.000000],[0,0,-1,0],[9E+09,9E+09,9E+09,9E+09,9E+09,9E+09]];
    CONST robtarget T1129:=[[64.000042,76.890746,9.749701],[1.000000,0.000000,0.000000,0.000000],[0,0,-1,0],[9E+09,9E+09,9E+09,9E+09,9E+09,9E+09]];
    CONST robtarget T1130:=[[62.500036,77.415670,9.749701],[1.000000,0.000000,0.000000,0.000000],[0,0,-1,0],[9E+09,9E+09,9E+09,9E+09,9E+09,9E+09]];
    CONST robtarget T1131:=[[62.500036,33.641491,9.749701],[1.000000,0.000000,0.000000,0.000000],[0,0,-1,0],[9E+09,9E+09,9E+09,9E+09,9E+09,9E+09]];
    CONST robtarget T1132:=[[61.000030,33.499307,9.749701],[1.000000,0.000000,0.000000,0.000000],[0,0,-1,0],[9E+09,9E+09,9E+09,9E+09,9E+09,9E+09]];
    CONST robtarget T1133:=[[61.000030,77.713251,9.749701],[1.000000,0.000000,0.000000,0.000000],[0,0,-1,0],[9E+09,9E+09,9E+09,9E+09,9E+09,9E+09]];
    CONST robtarget T1134:=[[59.500024,77.973848,9.749701],[1.000000,0.000000,0.000000,0.000000],[0,0,-1,0],[9E+09,9E+09,9E+09,9E+09,9E+09,9E+09]];
    CONST robtarget T1135:=[[59.500024,33.370393,9.749701],[1.000000,0.000000,0.000000,0.000000],[0,0,-1,0],[9E+09,9E+09,9E+09,9E+09,9E+09,9E+09]];
    CONST robtarget T1136:=[[58.000018,33.300180,9.749701],[1.000000,0.000000,0.000000,0.000000],[0,0,-1,0],[9E+09,9E+09,9E+09,9E+09,9E+09,9E+09]];
    CONST robtarget T1137:=[[58.000018,78.135313,9.749701],[1.000000,0.000000,0.000000,0.000000],[0,0,-1,0],[9E+09,9E+09,9E+09,9E+09,9E+09,9E+09]];
    CONST robtarget T1138:=[[56.500012,78.334377,9.749701],[1.000000,0.000000,0.000000,0.000000],[0,0,-1,0],[9E+09,9E+09,9E+09,9E+09,9E+09,9E+09]];
    CONST robtarget T1139:=[[56.500012,33.261967,9.749701],[1.000000,0.000000,0.000000,0.000000],[0,0,-1,0],[9E+09,9E+09,9E+09,9E+09,9E+09,9E+09]];
    CONST robtarget T1140:=[[55.000006,33.255796,9.749701],[1.000000,0.000000,0.000000,0.000000],[0,0,-1,0],[9E+09,9E+09,9E+09,9E+09,9E+09,9E+09]];
    CONST robtarget T1141:=[[55.000006,78.490912,9.749701],[1.000000,0.000000,0.000000,0.000000],[0,0,-1,0],[9E+09,9E+09,9E+09,9E+09,9E+09,9E+09]];
    CONST robtarget T1142:=[[53.500000,78.334376,9.749701],[1.000000,0.000000,0.000000,0.000000],[0,0,-1,0],[9E+09,9E+09,9E+09,9E+09,9E+09,9E+09]];
    CONST robtarget T1143:=[[53.500000,33.261970,9.749701],[1.000000,0.000000,0.000000,0.000000],[0,0,-1,0],[9E+09,9E+09,9E+09,9E+09,9E+09,9E+09]];
    CONST robtarget T1144:=[[51.999994,33.300183,9.749701],[1.000000,0.000000,0.000000,0.000000],[0,0,-1,0],[9E+09,9E+09,9E+09,9E+09,9E+09,9E+09]];
    CONST robtarget T1145:=[[51.999994,78.135313,9.749701],[1.000000,0.000000,0.000000,0.000000],[0,0,-1,0],[9E+09,9E+09,9E+09,9E+09,9E+09,9E+09]];
    CONST robtarget T1146:=[[50.499988,77.973848,9.749701],[1.000000,0.000000,0.000000,0.000000],[0,0,-1,0],[9E+09,9E+09,9E+09,9E+09,9E+09,9E+09]];
    CONST robtarget T1147:=[[50.499988,33.370393,9.749701],[1.000000,0.000000,0.000000,0.000000],[0,0,-1,0],[9E+09,9E+09,9E+09,9E+09,9E+09,9E+09]];
    CONST robtarget T1148:=[[48.999982,33.499307,9.749701],[1.000000,0.000000,0.000000,0.000000],[0,0,-1,0],[9E+09,9E+09,9E+09,9E+09,9E+09,9E+09]];
    CONST robtarget T1149:=[[48.999982,77.713250,9.749701],[1.000000,0.000000,0.000000,0.000000],[0,0,-1,0],[9E+09,9E+09,9E+09,9E+09,9E+09,9E+09]];
    CONST robtarget T1150:=[[47.499976,77.415670,9.749701],[1.000000,0.000000,0.000000,0.000000],[0,0,-1,0],[9E+09,9E+09,9E+09,9E+09,9E+09,9E+09]];
    CONST robtarget T1151:=[[47.499976,33.641491,9.749701],[1.000000,0.000000,0.000000,0.000000],[0,0,-1,0],[9E+09,9E+09,9E+09,9E+09,9E+09,9E+09]];
    CONST robtarget T1152:=[[45.999970,33.935928,9.749701],[1.000000,0.000000,0.000000,0.000000],[0,0,-1,0],[9E+09,9E+09,9E+09,9E+09,9E+09,9E+09]];
    CONST robtarget T1153:=[[45.999970,76.890746,9.749701],[1.000000,0.000000,0.000000,0.000000],[0,0,-1,0],[9E+09,9E+09,9E+09,9E+09,9E+09,9E+09]];
    CONST robtarget T1154:=[[44.499964,76.161667,9.749701],[1.000000,0.000000,0.000000,0.000000],[0,0,-1,0],[9E+09,9E+09,9E+09,9E+09,9E+09,9E+09]];
    CONST robtarget T1155:=[[44.499964,34.259033,9.749701],[1.000000,0.000000,0.000000,0.000000],[0,0,-1,0],[9E+09,9E+09,9E+09,9E+09,9E+09,9E+09]];
    CONST robtarget T1156:=[[42.999958,34.820110,9.749701],[1.000000,0.000000,0.000000,0.000000],[0,0,-1,0],[9E+09,9E+09,9E+09,9E+09,9E+09,9E+09]];
    CONST robtarget T1157:=[[42.999958,75.188416,9.749701],[1.000000,0.000000,0.000000,0.000000],[0,0,-1,0],[9E+09,9E+09,9E+09,9E+09,9E+09,9E+09]];
    CONST robtarget T1158:=[[41.499952,73.885585,9.749701],[1.000000,0.000000,0.000000,0.000000],[0,0,-1,0],[9E+09,9E+09,9E+09,9E+09,9E+09,9E+09]];
    CONST robtarget T1159:=[[41.499952,35.435172,9.749701],[1.000000,0.000000,0.000000,0.000000],[0,0,-1,0],[9E+09,9E+09,9E+09,9E+09,9E+09,9E+09]];
    CONST robtarget T1160:=[[39.999946,36.281324,9.749701],[1.000000,0.000000,0.000000,0.000000],[0,0,-1,0],[9E+09,9E+09,9E+09,9E+09,9E+09,9E+09]];
    CONST robtarget T1161:=[[39.999946,72.149604,9.749701],[1.000000,0.000000,0.000000,0.000000],[0,0,-1,0],[9E+09,9E+09,9E+09,9E+09,9E+09,9E+09]];
    CONST robtarget T1162:=[[38.499940,70.071652,9.749701],[1.000000,0.000000,0.000000,0.000000],[0,0,-1,0],[9E+09,9E+09,9E+09,9E+09,9E+09,9E+09]];
    CONST robtarget T1163:=[[38.499940,37.213527,9.749701],[1.000000,0.000000,0.000000,0.000000],[0,0,-1,0],[9E+09,9E+09,9E+09,9E+09,9E+09,9E+09]];
    CONST robtarget T1164:=[[36.999934,38.386643,9.749701],[1.000000,0.000000,0.000000,0.000000],[0,0,-1,0],[9E+09,9E+09,9E+09,9E+09,9E+09,9E+09]];
    CONST robtarget T1165:=[[36.999934,67.906293,9.749701],[1.000000,0.000000,0.000000,0.000000],[0,0,-1,0],[9E+09,9E+09,9E+09,9E+09,9E+09,9E+09]];
    CONST robtarget T1166:=[[35.499928,66.564678,9.749701],[1.000000,0.000000,0.000000,0.000000],[0,0,-1,0],[9E+09,9E+09,9E+09,9E+09,9E+09,9E+09]];
    CONST robtarget T1167:=[[35.499928,39.769866,9.749701],[1.000000,0.000000,0.000000,0.000000],[0,0,-1,0],[9E+09,9E+09,9E+09,9E+09,9E+09,9E+09]];
    CONST robtarget T1168:=[[33.999922,41.553007,9.749701],[1.000000,0.000000,0.000000,0.000000],[0,0,-1,0],[9E+09,9E+09,9E+09,9E+09,9E+09,9E+09]];
    CONST robtarget T1169:=[[33.999922,65.718152,9.749701],[1.000000,0.000000,0.000000,0.000000],[0,0,-1,0],[9E+09,9E+09,9E+09,9E+09,9E+09,9E+09]];
    CONST robtarget T1170:=[[32.499916,62.225279,9.749701],[1.000000,0.000000,0.000000,0.000000],[0,0,-1,0],[9E+09,9E+09,9E+09,9E+09,9E+09,9E+09]];
    CONST robtarget T1171:=[[32.499916,43.634111,9.749701],[1.000000,0.000000,0.000000,0.000000],[0,0,-1,0],[9E+09,9E+09,9E+09,9E+09,9E+09,9E+09]];
    CONST robtarget T1172:=[[30.999910,47.335884,9.749701],[1.000000,0.000000,0.000000,0.000000],[0,0,-1,0],[9E+09,9E+09,9E+09,9E+09,9E+09,9E+09]];
    CONST robtarget T1173:=[[30.999910,56.843137,9.749701],[1.000000,0.000000,0.000000,0.000000],[0,0,-1,0],[9E+09,9E+09,9E+09,9E+09,9E+09,9E+09]];
    CONST robtarget T1174:=[[30.999910,46.792186,10.249711],[1.000000,0.000000,0.000000,0.000000],[0,0,-1,0],[9E+09,9E+09,9E+09,9E+09,9E+09,9E+09]];
    CONST robtarget T1175:=[[30.999910,57.115259,10.249711],[1.000000,0.000000,0.000000,0.000000],[0,0,-1,0],[9E+09,9E+09,9E+09,9E+09,9E+09,9E+09]];
    CONST robtarget T1176:=[[30.999910,46.792186,10.249711],[1.000000,0.000000,0.000000,0.000000],[0,0,-1,0],[9E+09,9E+09,9E+09,9E+09,9E+09,9E+09]];
    CONST robtarget T1177:=[[30.999910,57.115259,10.249711],[1.000000,0.000000,0.000000,0.000000],[0,0,-1,0],[9E+09,9E+09,9E+09,9E+09,9E+09,9E+09]];
    CONST robtarget T1178:=[[32.499916,62.420969,10.249711],[1.000000,0.000000,0.000000,0.000000],[0,0,-1,0],[9E+09,9E+09,9E+09,9E+09,9E+09,9E+09]];
    CONST robtarget T1179:=[[32.499916,43.252123,10.249711],[1.000000,0.000000,0.000000,0.000000],[0,0,-1,0],[9E+09,9E+09,9E+09,9E+09,9E+09,9E+09]];
    CONST robtarget T1180:=[[33.999922,41.203816,10.249711],[1.000000,0.000000,0.000000,0.000000],[0,0,-1,0],[9E+09,9E+09,9E+09,9E+09,9E+09,9E+09]];
    CONST robtarget T1181:=[[33.999922,66.248963,10.249711],[1.000000,0.000000,0.000000,0.000000],[0,0,-1,0],[9E+09,9E+09,9E+09,9E+09,9E+09,9E+09]];
    CONST robtarget T1182:=[[35.499928,67.902618,10.249711],[1.000000,0.000000,0.000000,0.000000],[0,0,-1,0],[9E+09,9E+09,9E+09,9E+09,9E+09,9E+09]];
    CONST robtarget T1183:=[[35.499928,39.469911,10.249711],[1.000000,0.000000,0.000000,0.000000],[0,0,-1,0],[9E+09,9E+09,9E+09,9E+09,9E+09,9E+09]];
    CONST robtarget T1184:=[[36.999934,38.082377,10.249711],[1.000000,0.000000,0.000000,0.000000],[0,0,-1,0],[9E+09,9E+09,9E+09,9E+09,9E+09,9E+09]];
    CONST robtarget T1185:=[[36.999934,67.913115,10.249711],[1.000000,0.000000,0.000000,0.000000],[0,0,-1,0],[9E+09,9E+09,9E+09,9E+09,9E+09,9E+09]];
    CONST robtarget T1186:=[[38.499940,70.107722,10.249711],[1.000000,0.000000,0.000000,0.000000],[0,0,-1,0],[9E+09,9E+09,9E+09,9E+09,9E+09,9E+09]];
    CONST robtarget T1187:=[[38.499940,36.922147,10.249711],[1.000000,0.000000,0.000000,0.000000],[0,0,-1,0],[9E+09,9E+09,9E+09,9E+09,9E+09,9E+09]];
    CONST robtarget T1188:=[[39.999946,35.993646,10.249711],[1.000000,0.000000,0.000000,0.000000],[0,0,-1,0],[9E+09,9E+09,9E+09,9E+09,9E+09,9E+09]];
    CONST robtarget T1189:=[[39.999946,72.224497,10.249711],[1.000000,0.000000,0.000000,0.000000],[0,0,-1,0],[9E+09,9E+09,9E+09,9E+09,9E+09,9E+09]];
    CONST robtarget T1190:=[[41.499952,73.996171,10.249711],[1.000000,0.000000,0.000000,0.000000],[0,0,-1,0],[9E+09,9E+09,9E+09,9E+09,9E+09,9E+09]];
    CONST robtarget T1191:=[[41.499952,35.162754,10.249711],[1.000000,0.000000,0.000000,0.000000],[0,0,-1,0],[9E+09,9E+09,9E+09,9E+09,9E+09,9E+09]];
    CONST robtarget T1192:=[[42.999958,34.547692,10.249711],[1.000000,0.000000,0.000000,0.000000],[0,0,-1,0],[9E+09,9E+09,9E+09,9E+09,9E+09,9E+09]];
    CONST robtarget T1193:=[[42.999958,75.317084,10.249711],[1.000000,0.000000,0.000000,0.000000],[0,0,-1,0],[9E+09,9E+09,9E+09,9E+09,9E+09,9E+09]];
    CONST robtarget T1194:=[[44.499964,76.299782,10.249711],[1.000000,0.000000,0.000000,0.000000],[0,0,-1,0],[9E+09,9E+09,9E+09,9E+09,9E+09,9E+09]];
    CONST robtarget T1195:=[[44.499964,33.991774,10.249711],[1.000000,0.000000,0.000000,0.000000],[0,0,-1,0],[9E+09,9E+09,9E+09,9E+09,9E+09,9E+09]];
    CONST robtarget T1196:=[[45.999970,33.672314,10.249711],[1.000000,0.000000,0.000000,0.000000],[0,0,-1,0],[9E+09,9E+09,9E+09,9E+09,9E+09,9E+09]];
    CONST robtarget T1197:=[[45.999970,77.039357,10.249711],[1.000000,0.000000,0.000000,0.000000],[0,0,-1,0],[9E+09,9E+09,9E+09,9E+09,9E+09,9E+09]];
    CONST robtarget T1198:=[[47.499976,77.564206,10.249711],[1.000000,0.000000,0.000000,0.000000],[0,0,-1,0],[9E+09,9E+09,9E+09,9E+09,9E+09,9E+09]];
    CONST robtarget T1199:=[[47.499976,33.377658,10.249711],[1.000000,0.000000,0.000000,0.000000],[0,0,-1,0],[9E+09,9E+09,9E+09,9E+09,9E+09,9E+09]];
    CONST robtarget T1200:=[[48.999982,33.235474,10.249711],[1.000000,0.000000,0.000000,0.000000],[0,0,-1,0],[9E+09,9E+09,9E+09,9E+09,9E+09,9E+09]];
    CONST robtarget T1201:=[[48.999982,77.885457,10.249711],[1.000000,0.000000,0.000000,0.000000],[0,0,-1,0],[9E+09,9E+09,9E+09,9E+09,9E+09,9E+09]];
    CONST robtarget T1202:=[[50.499988,78.149918,10.249711],[1.000000,0.000000,0.000000,0.000000],[0,0,-1,0],[9E+09,9E+09,9E+09,9E+09,9E+09,9E+09]];
    CONST robtarget T1203:=[[50.499988,33.110183,10.249711],[1.000000,0.000000,0.000000,0.000000],[0,0,-1,0],[9E+09,9E+09,9E+09,9E+09,9E+09,9E+09]];
    CONST robtarget T1204:=[[51.999994,33.038234,10.249711],[1.000000,0.000000,0.000000,0.000000],[0,0,-1,0],[9E+09,9E+09,9E+09,9E+09,9E+09,9E+09]];
    CONST robtarget T1205:=[[51.999994,78.320464,10.249711],[1.000000,0.000000,0.000000,0.000000],[0,0,-1,0],[9E+09,9E+09,9E+09,9E+09,9E+09,9E+09]];
    CONST robtarget T1206:=[[53.500000,78.526703,10.249711],[1.000000,0.000000,0.000000,0.000000],[0,0,-1,0],[9E+09,9E+09,9E+09,9E+09,9E+09,9E+09]];
    CONST robtarget T1207:=[[53.500000,32.999779,10.249711],[1.000000,0.000000,0.000000,0.000000],[0,0,-1,0],[9E+09,9E+09,9E+09,9E+09,9E+09,9E+09]];
    CONST robtarget T1208:=[[55.000006,32.989987,10.249711],[1.000000,0.000000,0.000000,0.000000],[0,0,-1,0],[9E+09,9E+09,9E+09,9E+09,9E+09,9E+09]];
    CONST robtarget T1209:=[[55.000006,78.687676,10.249711],[1.000000,0.000000,0.000000,0.000000],[0,0,-1,0],[9E+09,9E+09,9E+09,9E+09,9E+09,9E+09]];
    CONST robtarget T1210:=[[56.500012,78.526704,10.249711],[1.000000,0.000000,0.000000,0.000000],[0,0,-1,0],[9E+09,9E+09,9E+09,9E+09,9E+09,9E+09]];
    CONST robtarget T1211:=[[56.500012,32.999776,10.249711],[1.000000,0.000000,0.000000,0.000000],[0,0,-1,0],[9E+09,9E+09,9E+09,9E+09,9E+09,9E+09]];
    CONST robtarget T1212:=[[58.000018,33.038230,10.249711],[1.000000,0.000000,0.000000,0.000000],[0,0,-1,0],[9E+09,9E+09,9E+09,9E+09,9E+09,9E+09]];
    CONST robtarget T1213:=[[58.000018,78.320464,10.249711],[1.000000,0.000000,0.000000,0.000000],[0,0,-1,0],[9E+09,9E+09,9E+09,9E+09,9E+09,9E+09]];
    CONST robtarget T1214:=[[59.500024,78.149918,10.249711],[1.000000,0.000000,0.000000,0.000000],[0,0,-1,0],[9E+09,9E+09,9E+09,9E+09,9E+09,9E+09]];
    CONST robtarget T1215:=[[59.500024,33.110183,10.249711],[1.000000,0.000000,0.000000,0.000000],[0,0,-1,0],[9E+09,9E+09,9E+09,9E+09,9E+09,9E+09]];
    CONST robtarget T1216:=[[61.000030,33.235474,10.249711],[1.000000,0.000000,0.000000,0.000000],[0,0,-1,0],[9E+09,9E+09,9E+09,9E+09,9E+09,9E+09]];
    CONST robtarget T1217:=[[61.000030,77.885457,10.249711],[1.000000,0.000000,0.000000,0.000000],[0,0,-1,0],[9E+09,9E+09,9E+09,9E+09,9E+09,9E+09]];
    CONST robtarget T1218:=[[62.500036,77.564206,10.249711],[1.000000,0.000000,0.000000,0.000000],[0,0,-1,0],[9E+09,9E+09,9E+09,9E+09,9E+09,9E+09]];
    CONST robtarget T1219:=[[62.500036,33.377658,10.249711],[1.000000,0.000000,0.000000,0.000000],[0,0,-1,0],[9E+09,9E+09,9E+09,9E+09,9E+09,9E+09]];
    CONST robtarget T1220:=[[64.000042,33.672314,10.249711],[1.000000,0.000000,0.000000,0.000000],[0,0,-1,0],[9E+09,9E+09,9E+09,9E+09,9E+09,9E+09]];
    CONST robtarget T1221:=[[64.000042,77.039357,10.249711],[1.000000,0.000000,0.000000,0.000000],[0,0,-1,0],[9E+09,9E+09,9E+09,9E+09,9E+09,9E+09]];
    CONST robtarget T1222:=[[65.500048,76.299783,10.249711],[1.000000,0.000000,0.000000,0.000000],[0,0,-1,0],[9E+09,9E+09,9E+09,9E+09,9E+09,9E+09]];
    CONST robtarget T1223:=[[65.500048,33.991773,10.249711],[1.000000,0.000000,0.000000,0.000000],[0,0,-1,0],[9E+09,9E+09,9E+09,9E+09,9E+09,9E+09]];
    CONST robtarget T1224:=[[67.000054,34.547694,10.249711],[1.000000,0.000000,0.000000,0.000000],[0,0,-1,0],[9E+09,9E+09,9E+09,9E+09,9E+09,9E+09]];
    CONST robtarget T1225:=[[67.000054,75.317086,10.249711],[1.000000,0.000000,0.000000,0.000000],[0,0,-1,0],[9E+09,9E+09,9E+09,9E+09,9E+09,9E+09]];
    CONST robtarget T1226:=[[68.500060,73.996173,10.249711],[1.000000,0.000000,0.000000,0.000000],[0,0,-1,0],[9E+09,9E+09,9E+09,9E+09,9E+09,9E+09]];
    CONST robtarget T1227:=[[68.500060,35.162762,10.249711],[1.000000,0.000000,0.000000,0.000000],[0,0,-1,0],[9E+09,9E+09,9E+09,9E+09,9E+09,9E+09]];
    CONST robtarget T1228:=[[70.000066,35.993653,10.249711],[1.000000,0.000000,0.000000,0.000000],[0,0,-1,0],[9E+09,9E+09,9E+09,9E+09,9E+09,9E+09]];
    CONST robtarget T1229:=[[70.000066,72.224499,10.249711],[1.000000,0.000000,0.000000,0.000000],[0,0,-1,0],[9E+09,9E+09,9E+09,9E+09,9E+09,9E+09]];
    CONST robtarget T1230:=[[71.500072,70.107724,10.249711],[1.000000,0.000000,0.000000,0.000000],[0,0,-1,0],[9E+09,9E+09,9E+09,9E+09,9E+09,9E+09]];
    CONST robtarget T1231:=[[71.500072,36.922147,10.249711],[1.000000,0.000000,0.000000,0.000000],[0,0,-1,0],[9E+09,9E+09,9E+09,9E+09,9E+09,9E+09]];
    CONST robtarget T1232:=[[73.000078,38.082376,10.249711],[1.000000,0.000000,0.000000,0.000000],[0,0,-1,0],[9E+09,9E+09,9E+09,9E+09,9E+09,9E+09]];
    CONST robtarget T1233:=[[73.000078,67.912749,10.249711],[1.000000,0.000000,0.000000,0.000000],[0,0,-1,0],[9E+09,9E+09,9E+09,9E+09,9E+09,9E+09]];
    CONST robtarget T1234:=[[74.500084,67.902606,10.249711],[1.000000,0.000000,0.000000,0.000000],[0,0,-1,0],[9E+09,9E+09,9E+09,9E+09,9E+09,9E+09]];
    CONST robtarget T1235:=[[74.500084,39.469910,10.249711],[1.000000,0.000000,0.000000,0.000000],[0,0,-1,0],[9E+09,9E+09,9E+09,9E+09,9E+09,9E+09]];
    CONST robtarget T1236:=[[76.000090,41.203814,10.249711],[1.000000,0.000000,0.000000,0.000000],[0,0,-1,0],[9E+09,9E+09,9E+09,9E+09,9E+09,9E+09]];
    CONST robtarget T1237:=[[76.000090,66.249074,10.249711],[1.000000,0.000000,0.000000,0.000000],[0,0,-1,0],[9E+09,9E+09,9E+09,9E+09,9E+09,9E+09]];
    CONST robtarget T1238:=[[77.500096,62.418544,10.249711],[1.000000,0.000000,0.000000,0.000000],[0,0,-1,0],[9E+09,9E+09,9E+09,9E+09,9E+09,9E+09]];
    CONST robtarget T1239:=[[77.500096,43.252118,10.249711],[1.000000,0.000000,0.000000,0.000000],[0,0,-1,0],[9E+09,9E+09,9E+09,9E+09,9E+09,9E+09]];
    CONST robtarget T1240:=[[79.000102,46.792179,10.249711],[1.000000,0.000000,0.000000,0.000000],[0,0,-1,0],[9E+09,9E+09,9E+09,9E+09,9E+09,9E+09]];
    CONST robtarget T1241:=[[79.000102,57.114614,10.249711],[1.000000,0.000000,0.000000,0.000000],[0,0,-1,0],[9E+09,9E+09,9E+09,9E+09,9E+09,9E+09]];
    CONST robtarget T1242:=[[79.000102,46.450116,10.749721],[1.000000,0.000000,0.000000,0.000000],[0,0,-1,0],[9E+09,9E+09,9E+09,9E+09,9E+09,9E+09]];
    CONST robtarget T1243:=[[79.000102,57.380675,10.749721],[1.000000,0.000000,0.000000,0.000000],[0,0,-1,0],[9E+09,9E+09,9E+09,9E+09,9E+09,9E+09]];
    CONST robtarget T1244:=[[79.000102,46.450116,10.749721],[1.000000,0.000000,0.000000,0.000000],[0,0,-1,0],[9E+09,9E+09,9E+09,9E+09,9E+09,9E+09]];
    CONST robtarget T1245:=[[79.000102,57.380675,10.749721],[1.000000,0.000000,0.000000,0.000000],[0,0,-1,0],[9E+09,9E+09,9E+09,9E+09,9E+09,9E+09]];
    CONST robtarget T1246:=[[77.500096,62.575091,10.749721],[1.000000,0.000000,0.000000,0.000000],[0,0,-1,0],[9E+09,9E+09,9E+09,9E+09,9E+09,9E+09]];
    CONST robtarget T1247:=[[77.500096,42.929365,10.749721],[1.000000,0.000000,0.000000,0.000000],[0,0,-1,0],[9E+09,9E+09,9E+09,9E+09,9E+09,9E+09]];
    CONST robtarget T1248:=[[76.000090,40.866390,10.749721],[1.000000,0.000000,0.000000,0.000000],[0,0,-1,0],[9E+09,9E+09,9E+09,9E+09,9E+09,9E+09]];
    CONST robtarget T1249:=[[76.000090,66.632607,10.749721],[1.000000,0.000000,0.000000,0.000000],[0,0,-1,0],[9E+09,9E+09,9E+09,9E+09,9E+09,9E+09]];
    CONST robtarget T1250:=[[74.500084,68.504039,10.749721],[1.000000,0.000000,0.000000,0.000000],[0,0,-1,0],[9E+09,9E+09,9E+09,9E+09,9E+09,9E+09]];
    CONST robtarget T1251:=[[74.500084,39.169955,10.749721],[1.000000,0.000000,0.000000,0.000000],[0,0,-1,0],[9E+09,9E+09,9E+09,9E+09,9E+09,9E+09]];
    CONST robtarget T1252:=[[73.000078,37.782421,10.749721],[1.000000,0.000000,0.000000,0.000000],[0,0,-1,0],[9E+09,9E+09,9E+09,9E+09,9E+09,9E+09]];
    CONST robtarget T1253:=[[73.000078,67.919623,10.749721],[1.000000,0.000000,0.000000,0.000000],[0,0,-1,0],[9E+09,9E+09,9E+09,9E+09,9E+09,9E+09]];
    CONST robtarget T1254:=[[71.500072,70.143795,10.749721],[1.000000,0.000000,0.000000,0.000000],[0,0,-1,0],[9E+09,9E+09,9E+09,9E+09,9E+09,9E+09]];
    CONST robtarget T1255:=[[71.500072,36.634471,10.749721],[1.000000,0.000000,0.000000,0.000000],[0,0,-1,0],[9E+09,9E+09,9E+09,9E+09,9E+09,9E+09]];
    CONST robtarget T1256:=[[70.000066,35.705977,10.749721],[1.000000,0.000000,0.000000,0.000000],[0,0,-1,0],[9E+09,9E+09,9E+09,9E+09,9E+09,9E+09]];
    CONST robtarget T1257:=[[70.000066,72.299392,10.749721],[1.000000,0.000000,0.000000,0.000000],[0,0,-1,0],[9E+09,9E+09,9E+09,9E+09,9E+09,9E+09]];
    CONST robtarget T1258:=[[68.500060,74.106760,10.749721],[1.000000,0.000000,0.000000,0.000000],[0,0,-1,0],[9E+09,9E+09,9E+09,9E+09,9E+09,9E+09]];
    CONST robtarget T1259:=[[68.500060,34.890346,10.749721],[1.000000,0.000000,0.000000,0.000000],[0,0,-1,0],[9E+09,9E+09,9E+09,9E+09,9E+09,9E+09]];
    CONST robtarget T1260:=[[67.000054,34.287111,10.749721],[1.000000,0.000000,0.000000,0.000000],[0,0,-1,0],[9E+09,9E+09,9E+09,9E+09,9E+09,9E+09]];
    CONST robtarget T1261:=[[67.000054,75.449229,10.749721],[1.000000,0.000000,0.000000,0.000000],[0,0,-1,0],[9E+09,9E+09,9E+09,9E+09,9E+09,9E+09]];
    CONST robtarget T1262:=[[65.500048,76.431573,10.749721],[1.000000,0.000000,0.000000,0.000000],[0,0,-1,0],[9E+09,9E+09,9E+09,9E+09,9E+09,9E+09]];
    CONST robtarget T1263:=[[65.500048,33.765589,10.749721],[1.000000,0.000000,0.000000,0.000000],[0,0,-1,0],[9E+09,9E+09,9E+09,9E+09,9E+09,9E+09]];
    CONST robtarget T1264:=[[64.000042,33.445948,10.749721],[1.000000,0.000000,0.000000,0.000000],[0,0,-1,0],[9E+09,9E+09,9E+09,9E+09,9E+09,9E+09]];
    CONST robtarget T1265:=[[64.000042,77.187968,10.749721],[1.000000,0.000000,0.000000,0.000000],[0,0,-1,0],[9E+09,9E+09,9E+09,9E+09,9E+09,9E+09]];
    CONST robtarget T1266:=[[62.500036,77.712750,10.749721],[1.000000,0.000000,0.000000,0.000000],[0,0,-1,0],[9E+09,9E+09,9E+09,9E+09,9E+09,9E+09]];
    CONST robtarget T1267:=[[62.500036,33.150426,10.749721],[1.000000,0.000000,0.000000,0.000000],[0,0,-1,0],[9E+09,9E+09,9E+09,9E+09,9E+09,9E+09]];
    CONST robtarget T1268:=[[61.000030,33.007847,10.749721],[1.000000,0.000000,0.000000,0.000000],[0,0,-1,0],[9E+09,9E+09,9E+09,9E+09,9E+09,9E+09]];
    CONST robtarget T1269:=[[61.000030,78.057664,10.749721],[1.000000,0.000000,0.000000,0.000000],[0,0,-1,0],[9E+09,9E+09,9E+09,9E+09,9E+09,9E+09]];
    CONST robtarget T1270:=[[59.500024,78.325988,10.749721],[1.000000,0.000000,0.000000,0.000000],[0,0,-1,0],[9E+09,9E+09,9E+09,9E+09,9E+09,9E+09]];
    CONST robtarget T1271:=[[59.500024,32.879920,10.749721],[1.000000,0.000000,0.000000,0.000000],[0,0,-1,0],[9E+09,9E+09,9E+09,9E+09,9E+09,9E+09]];
    CONST robtarget T1272:=[[58.000018,32.804536,10.749721],[1.000000,0.000000,0.000000,0.000000],[0,0,-1,0],[9E+09,9E+09,9E+09,9E+09,9E+09,9E+09]];
    CONST robtarget T1273:=[[58.000018,78.505615,10.749721],[1.000000,0.000000,0.000000,0.000000],[0,0,-1,0],[9E+09,9E+09,9E+09,9E+09,9E+09,9E+09]];
    CONST robtarget T1274:=[[56.500012,78.719031,10.749721],[1.000000,0.000000,0.000000,0.000000],[0,0,-1,0],[9E+09,9E+09,9E+09,9E+09,9E+09,9E+09]];
    CONST robtarget T1275:=[[56.500012,32.758484,10.749721],[1.000000,0.000000,0.000000,0.000000],[0,0,-1,0],[9E+09,9E+09,9E+09,9E+09,9E+09,9E+09]];
    CONST robtarget T1276:=[[55.000006,32.734943,10.749721],[1.000000,0.000000,0.000000,0.000000],[0,0,-1,0],[9E+09,9E+09,9E+09,9E+09,9E+09,9E+09]];
    CONST robtarget T1277:=[[55.000006,78.884440,10.749721],[1.000000,0.000000,0.000000,0.000000],[0,0,-1,0],[9E+09,9E+09,9E+09,9E+09,9E+09,9E+09]];
    CONST robtarget T1278:=[[53.500000,78.719030,10.749721],[1.000000,0.000000,0.000000,0.000000],[0,0,-1,0],[9E+09,9E+09,9E+09,9E+09,9E+09,9E+09]];
    CONST robtarget T1279:=[[53.500000,32.758486,10.749721],[1.000000,0.000000,0.000000,0.000000],[0,0,-1,0],[9E+09,9E+09,9E+09,9E+09,9E+09,9E+09]];
    CONST robtarget T1280:=[[51.999994,32.804538,10.749721],[1.000000,0.000000,0.000000,0.000000],[0,0,-1,0],[9E+09,9E+09,9E+09,9E+09,9E+09,9E+09]];
    CONST robtarget T1281:=[[51.999994,78.505615,10.749721],[1.000000,0.000000,0.000000,0.000000],[0,0,-1,0],[9E+09,9E+09,9E+09,9E+09,9E+09,9E+09]];
    CONST robtarget T1282:=[[50.499988,78.325988,10.749721],[1.000000,0.000000,0.000000,0.000000],[0,0,-1,0],[9E+09,9E+09,9E+09,9E+09,9E+09,9E+09]];
    CONST robtarget T1283:=[[50.499988,32.879920,10.749721],[1.000000,0.000000,0.000000,0.000000],[0,0,-1,0],[9E+09,9E+09,9E+09,9E+09,9E+09,9E+09]];
    CONST robtarget T1284:=[[48.999982,33.007847,10.749721],[1.000000,0.000000,0.000000,0.000000],[0,0,-1,0],[9E+09,9E+09,9E+09,9E+09,9E+09,9E+09]];
    CONST robtarget T1285:=[[48.999982,78.057663,10.749721],[1.000000,0.000000,0.000000,0.000000],[0,0,-1,0],[9E+09,9E+09,9E+09,9E+09,9E+09,9E+09]];
    CONST robtarget T1286:=[[47.499976,77.712750,10.749721],[1.000000,0.000000,0.000000,0.000000],[0,0,-1,0],[9E+09,9E+09,9E+09,9E+09,9E+09,9E+09]];
    CONST robtarget T1287:=[[47.499976,33.150427,10.749721],[1.000000,0.000000,0.000000,0.000000],[0,0,-1,0],[9E+09,9E+09,9E+09,9E+09,9E+09,9E+09]];
    CONST robtarget T1288:=[[45.999970,33.445949,10.749721],[1.000000,0.000000,0.000000,0.000000],[0,0,-1,0],[9E+09,9E+09,9E+09,9E+09,9E+09,9E+09]];
    CONST robtarget T1289:=[[45.999970,77.187967,10.749721],[1.000000,0.000000,0.000000,0.000000],[0,0,-1,0],[9E+09,9E+09,9E+09,9E+09,9E+09,9E+09]];
    CONST robtarget T1290:=[[44.499964,76.431571,10.749721],[1.000000,0.000000,0.000000,0.000000],[0,0,-1,0],[9E+09,9E+09,9E+09,9E+09,9E+09,9E+09]];
    CONST robtarget T1291:=[[44.499964,33.765590,10.749721],[1.000000,0.000000,0.000000,0.000000],[0,0,-1,0],[9E+09,9E+09,9E+09,9E+09,9E+09,9E+09]];
    CONST robtarget T1292:=[[42.999958,34.287108,10.749721],[1.000000,0.000000,0.000000,0.000000],[0,0,-1,0],[9E+09,9E+09,9E+09,9E+09,9E+09,9E+09]];
    CONST robtarget T1293:=[[42.999958,75.449227,10.749721],[1.000000,0.000000,0.000000,0.000000],[0,0,-1,0],[9E+09,9E+09,9E+09,9E+09,9E+09,9E+09]];
    CONST robtarget T1294:=[[41.499952,74.106757,10.749721],[1.000000,0.000000,0.000000,0.000000],[0,0,-1,0],[9E+09,9E+09,9E+09,9E+09,9E+09,9E+09]];
    CONST robtarget T1295:=[[41.499952,34.890336,10.749721],[1.000000,0.000000,0.000000,0.000000],[0,0,-1,0],[9E+09,9E+09,9E+09,9E+09,9E+09,9E+09]];
    CONST robtarget T1296:=[[39.999946,35.705967,10.749721],[1.000000,0.000000,0.000000,0.000000],[0,0,-1,0],[9E+09,9E+09,9E+09,9E+09,9E+09,9E+09]];
    CONST robtarget T1297:=[[39.999946,72.299389,10.749721],[1.000000,0.000000,0.000000,0.000000],[0,0,-1,0],[9E+09,9E+09,9E+09,9E+09,9E+09,9E+09]];
    CONST robtarget T1298:=[[38.499940,70.143791,10.749721],[1.000000,0.000000,0.000000,0.000000],[0,0,-1,0],[9E+09,9E+09,9E+09,9E+09,9E+09,9E+09]];
    CONST robtarget T1299:=[[38.499940,36.634469,10.749721],[1.000000,0.000000,0.000000,0.000000],[0,0,-1,0],[9E+09,9E+09,9E+09,9E+09,9E+09,9E+09]];
    CONST robtarget T1300:=[[36.999934,37.782423,10.749721],[1.000000,0.000000,0.000000,0.000000],[0,0,-1,0],[9E+09,9E+09,9E+09,9E+09,9E+09,9E+09]];
    CONST robtarget T1301:=[[36.999934,67.919936,10.749721],[1.000000,0.000000,0.000000,0.000000],[0,0,-1,0],[9E+09,9E+09,9E+09,9E+09,9E+09,9E+09]];
    CONST robtarget T1302:=[[35.499928,68.504037,10.749721],[1.000000,0.000000,0.000000,0.000000],[0,0,-1,0],[9E+09,9E+09,9E+09,9E+09,9E+09,9E+09]];
    CONST robtarget T1303:=[[35.499928,39.169957,10.749721],[1.000000,0.000000,0.000000,0.000000],[0,0,-1,0],[9E+09,9E+09,9E+09,9E+09,9E+09,9E+09]];
    CONST robtarget T1304:=[[33.999922,40.866394,10.749721],[1.000000,0.000000,0.000000,0.000000],[0,0,-1,0],[9E+09,9E+09,9E+09,9E+09,9E+09,9E+09]];
    CONST robtarget T1305:=[[33.999922,66.632876,10.749721],[1.000000,0.000000,0.000000,0.000000],[0,0,-1,0],[9E+09,9E+09,9E+09,9E+09,9E+09,9E+09]];
    CONST robtarget T1306:=[[32.499916,62.575250,10.749721],[1.000000,0.000000,0.000000,0.000000],[0,0,-1,0],[9E+09,9E+09,9E+09,9E+09,9E+09,9E+09]];
    CONST robtarget T1307:=[[32.499916,42.929371,10.749721],[1.000000,0.000000,0.000000,0.000000],[0,0,-1,0],[9E+09,9E+09,9E+09,9E+09,9E+09,9E+09]];
    CONST robtarget T1308:=[[30.999910,46.450123,10.749721],[1.000000,0.000000,0.000000,0.000000],[0,0,-1,0],[9E+09,9E+09,9E+09,9E+09,9E+09,9E+09]];
    CONST robtarget T1309:=[[30.999910,57.378980,10.749721],[1.000000,0.000000,0.000000,0.000000],[0,0,-1,0],[9E+09,9E+09,9E+09,9E+09,9E+09,9E+09]];
    CONST robtarget T1310:=[[30.999910,46.435801,11.249731],[1.000000,0.000000,0.000000,0.000000],[0,0,-1,0],[9E+09,9E+09,9E+09,9E+09,9E+09,9E+09]];
    CONST robtarget T1311:=[[30.999910,57.642704,11.249731],[1.000000,0.000000,0.000000,0.000000],[0,0,-1,0],[9E+09,9E+09,9E+09,9E+09,9E+09,9E+09]];
    CONST robtarget T1312:=[[30.999910,46.435801,11.249731],[1.000000,0.000000,0.000000,0.000000],[0,0,-1,0],[9E+09,9E+09,9E+09,9E+09,9E+09,9E+09]];
    CONST robtarget T1313:=[[30.999910,57.642704,11.249731],[1.000000,0.000000,0.000000,0.000000],[0,0,-1,0],[9E+09,9E+09,9E+09,9E+09,9E+09,9E+09]];
    CONST robtarget T1314:=[[32.499916,62.697592,11.249731],[1.000000,0.000000,0.000000,0.000000],[0,0,-1,0],[9E+09,9E+09,9E+09,9E+09,9E+09,9E+09]];
    CONST robtarget T1315:=[[32.499916,42.884164,11.249731],[1.000000,0.000000,0.000000,0.000000],[0,0,-1,0],[9E+09,9E+09,9E+09,9E+09,9E+09,9E+09]];
    CONST robtarget T1316:=[[33.999922,40.749864,11.249731],[1.000000,0.000000,0.000000,0.000000],[0,0,-1,0],[9E+09,9E+09,9E+09,9E+09,9E+09,9E+09]];
    CONST robtarget T1317:=[[33.999922,66.711475,11.249731],[1.000000,0.000000,0.000000,0.000000],[0,0,-1,0],[9E+09,9E+09,9E+09,9E+09,9E+09,9E+09]];
    CONST robtarget T1318:=[[35.499928,68.889789,11.249731],[1.000000,0.000000,0.000000,0.000000],[0,0,-1,0],[9E+09,9E+09,9E+09,9E+09,9E+09,9E+09]];
    CONST robtarget T1319:=[[35.499928,39.061596,11.249731],[1.000000,0.000000,0.000000,0.000000],[0,0,-1,0],[9E+09,9E+09,9E+09,9E+09,9E+09,9E+09]];
    CONST robtarget T1320:=[[36.999934,37.663817,11.249731],[1.000000,0.000000,0.000000,0.000000],[0,0,-1,0],[9E+09,9E+09,9E+09,9E+09,9E+09,9E+09]];
    CONST robtarget T1321:=[[36.999934,67.926758,11.249731],[1.000000,0.000000,0.000000,0.000000],[0,0,-1,0],[9E+09,9E+09,9E+09,9E+09,9E+09,9E+09]];
    CONST robtarget T1322:=[[38.499940,70.176866,11.249731],[1.000000,0.000000,0.000000,0.000000],[0,0,-1,0],[9E+09,9E+09,9E+09,9E+09,9E+09,9E+09]];
    CONST robtarget T1323:=[[38.499940,36.498798,11.249731],[1.000000,0.000000,0.000000,0.000000],[0,0,-1,0],[9E+09,9E+09,9E+09,9E+09,9E+09,9E+09]];
    CONST robtarget T1324:=[[39.999946,35.561578,11.249731],[1.000000,0.000000,0.000000,0.000000],[0,0,-1,0],[9E+09,9E+09,9E+09,9E+09,9E+09,9E+09]];
    CONST robtarget T1325:=[[39.999946,72.359453,11.249731],[1.000000,0.000000,0.000000,0.000000],[0,0,-1,0],[9E+09,9E+09,9E+09,9E+09,9E+09,9E+09]];
    CONST robtarget T1326:=[[41.499952,74.217344,11.249731],[1.000000,0.000000,0.000000,0.000000],[0,0,-1,0],[9E+09,9E+09,9E+09,9E+09,9E+09,9E+09]];
    CONST robtarget T1327:=[[41.499952,34.764679,11.249731],[1.000000,0.000000,0.000000,0.000000],[0,0,-1,0],[9E+09,9E+09,9E+09,9E+09,9E+09,9E+09]];
    CONST robtarget T1328:=[[42.999958,34.184980,11.249731],[1.000000,0.000000,0.000000,0.000000],[0,0,-1,0],[9E+09,9E+09,9E+09,9E+09,9E+09,9E+09]];
    CONST robtarget T1329:=[[42.999958,75.583686,11.249731],[1.000000,0.000000,0.000000,0.000000],[0,0,-1,0],[9E+09,9E+09,9E+09,9E+09,9E+09,9E+09]];
    CONST robtarget T1330:=[[44.499964,76.563361,11.249731],[1.000000,0.000000,0.000000,0.000000],[0,0,-1,0],[9E+09,9E+09,9E+09,9E+09,9E+09,9E+09]];
    CONST robtarget T1331:=[[44.499964,33.666327,11.249731],[1.000000,0.000000,0.000000,0.000000],[0,0,-1,0],[9E+09,9E+09,9E+09,9E+09,9E+09,9E+09]];
    CONST robtarget T1332:=[[45.999970,33.346033,11.249731],[1.000000,0.000000,0.000000,0.000000],[0,0,-1,0],[9E+09,9E+09,9E+09,9E+09,9E+09,9E+09]];
    CONST robtarget T1333:=[[45.999970,77.336578,11.249731],[1.000000,0.000000,0.000000,0.000000],[0,0,-1,0],[9E+09,9E+09,9E+09,9E+09,9E+09,9E+09]];
    CONST robtarget T1334:=[[47.499976,77.860099,11.249731],[1.000000,0.000000,0.000000,0.000000],[0,0,-1,0],[9E+09,9E+09,9E+09,9E+09,9E+09,9E+09]];
    CONST robtarget T1335:=[[47.499976,33.049486,11.249731],[1.000000,0.000000,0.000000,0.000000],[0,0,-1,0],[9E+09,9E+09,9E+09,9E+09,9E+09,9E+09]];
    CONST robtarget T1336:=[[48.999982,32.906907,11.249731],[1.000000,0.000000,0.000000,0.000000],[0,0,-1,0],[9E+09,9E+09,9E+09,9E+09,9E+09,9E+09]];
    CONST robtarget T1337:=[[48.999982,78.215623,11.249731],[1.000000,0.000000,0.000000,0.000000],[0,0,-1,0],[9E+09,9E+09,9E+09,9E+09,9E+09,9E+09]];
    CONST robtarget T1338:=[[50.499988,78.482418,11.249731],[1.000000,0.000000,0.000000,0.000000],[0,0,-1,0],[9E+09,9E+09,9E+09,9E+09,9E+09,9E+09]];
    CONST robtarget T1339:=[[50.499988,32.766519,11.249731],[1.000000,0.000000,0.000000,0.000000],[0,0,-1,0],[9E+09,9E+09,9E+09,9E+09,9E+09,9E+09]];
    CONST robtarget T1340:=[[51.999994,32.690375,11.249731],[1.000000,0.000000,0.000000,0.000000],[0,0,-1,0],[9E+09,9E+09,9E+09,9E+09,9E+09,9E+09]];
    CONST robtarget T1341:=[[51.999994,78.684281,11.249731],[1.000000,0.000000,0.000000,0.000000],[0,0,-1,0],[9E+09,9E+09,9E+09,9E+09,9E+09,9E+09]];
    CONST robtarget T1342:=[[53.500000,78.911358,11.249731],[1.000000,0.000000,0.000000,0.000000],[0,0,-1,0],[9E+09,9E+09,9E+09,9E+09,9E+09,9E+09]];
    CONST robtarget T1343:=[[53.500000,32.643954,11.249731],[1.000000,0.000000,0.000000,0.000000],[0,0,-1,0],[9E+09,9E+09,9E+09,9E+09,9E+09,9E+09]];
    CONST robtarget T1344:=[[55.000006,32.619365,11.249731],[1.000000,0.000000,0.000000,0.000000],[0,0,-1,0],[9E+09,9E+09,9E+09,9E+09,9E+09,9E+09]];
    CONST robtarget T1345:=[[55.000006,79.081205,11.249731],[1.000000,0.000000,0.000000,0.000000],[0,0,-1,0],[9E+09,9E+09,9E+09,9E+09,9E+09,9E+09]];
    CONST robtarget T1346:=[[56.500012,78.911358,11.249731],[1.000000,0.000000,0.000000,0.000000],[0,0,-1,0],[9E+09,9E+09,9E+09,9E+09,9E+09,9E+09]];
    CONST robtarget T1347:=[[56.500012,32.643952,11.249731],[1.000000,0.000000,0.000000,0.000000],[0,0,-1,0],[9E+09,9E+09,9E+09,9E+09,9E+09,9E+09]];
    CONST robtarget T1348:=[[58.000018,32.690373,11.249731],[1.000000,0.000000,0.000000,0.000000],[0,0,-1,0],[9E+09,9E+09,9E+09,9E+09,9E+09,9E+09]];
    CONST robtarget T1349:=[[58.000018,78.684282,11.249731],[1.000000,0.000000,0.000000,0.000000],[0,0,-1,0],[9E+09,9E+09,9E+09,9E+09,9E+09,9E+09]];
    CONST robtarget T1350:=[[59.500024,78.482418,11.249731],[1.000000,0.000000,0.000000,0.000000],[0,0,-1,0],[9E+09,9E+09,9E+09,9E+09,9E+09,9E+09]];
    CONST robtarget T1351:=[[59.500024,32.766519,11.249731],[1.000000,0.000000,0.000000,0.000000],[0,0,-1,0],[9E+09,9E+09,9E+09,9E+09,9E+09,9E+09]];
    CONST robtarget T1352:=[[61.000030,32.906907,11.249731],[1.000000,0.000000,0.000000,0.000000],[0,0,-1,0],[9E+09,9E+09,9E+09,9E+09,9E+09,9E+09]];
